LIN {X 0.125,Y -605.700,Z 1096.668,A 0.000,B 0.000,C 90.000,E1 336.230} C_DIS
LIN {X 0.154,Y -607.476,Z 1096.661,A 0.000,B 0.000,C 90.000,E1 334.921} C_DIS
LIN {X -0.038,Y -608.596,Z 1096.655,A 0.000,B 0.000,C 90.000,E1 333.896} C_DIS
LIN {X -0.170,Y -609.283,Z 1096.651,A 0.000,B 0.000,C 90.000,E1 333.127} C_DIS
LIN {X -0.338,Y -609.953,Z 1096.645,A 0.000,B 0.000,C 90.000,E1 332.103} C_DIS
LIN {X -0.253,Y -610.415,Z 1096.638,A 0.000,B 0.000,C 90.000,E1 330.795} C_DIS
LIN {X -0.035,Y -610.410,Z 1096.635,A 0.000,B 0.000,C 90.000,E1 330.255} C_DIS
LIN {X 0.098,Y -609.926,Z 1096.629,A 0.000,B 0.000,C 90.000,E1 329.203} C_DIS
LIN {X 0.317,Y -609.470,Z 1096.626,A 0.000,B 0.000,C 90.000,E1 328.663} C_DIS
LIN {X -0.091,Y -608.172,Z 1096.620,A 0.000,B 0.000,C 90.000,E1 327.661} C_DIS
LIN {X 0.115,Y -607.438,Z 1096.617,A 0.000,B 0.000,C 90.000,E1 327.120} C_DIS
LIN {X 0.003,Y -605.362,Z 1096.612,A 0.000,B 0.000,C 90.000,E1 326.087} C_DIS
LIN {X -0.052,Y -603.766,Z 1096.607,A 0.000,B 0.000,C 90.000,E1 325.308} C_DIS
LIN {X -0.119,Y -602.105,Z 1096.603,A 0.000,B 0.000,C 90.000,E1 324.529} C_DIS
LIN {X 0.286,Y -600.441,Z 1096.599,A 0.000,B 0.000,C 90.000,E1 323.703} C_DIS
LIN {X 0.181,Y -598.723,Z 1096.594,A 0.000,B 0.000,C 90.000,E1 322.924} C_DIS
LIN {X 0.050,Y -595.950,Z 1096.587,A 0.000,B 0.000,C 90.000,E1 321.618} C_DIS
LIN {X 0.006,Y -592.496,Z 1096.578,A 0.000,B 0.000,C 90.000,E1 320.033} C_DIS
LIN {X 0.147,Y -589.672,Z 1096.571,A 0.000,B 0.000,C 90.000,E1 318.690} C_DIS
LIN {X -0.213,Y -586.399,Z 1096.563,A 0.000,B 0.000,C 90.000,E1 317.391} C_DIS
LIN {X -0.034,Y -585.691,Z 1096.562,A 0.000,B 0.000,C 90.000,E1 317.106} C_DIS
LIN {X 0.326,Y -581.328,Z 1096.554,A 0.000,B 0.000,C 90.000,E1 315.729} C_DIS
LIN {X -0.064,Y -578.377,Z 1096.550,A 0.000,B 0.000,C 90.000,E1 314.960} C_DIS
LIN {X -0.234,Y -573.232,Z 1096.542,A 0.000,B 0.000,C 90.000,E1 313.623} C_DIS
LIN {X -0.007,Y -571.099,Z 1096.539,A 0.000,B 0.000,C 90.000,E1 313.056} C_DIS
LIN {X -0.067,Y -567.497,Z 1096.535,A 0.000,B 0.000,C 90.000,E1 312.243} C_DIS
LIN {X -0.132,Y -565.501,Z 1096.532,A 0.000,B 0.000,C 90.000,E1 311.838} C_DIS
LIN {X -0.012,Y -560.708,Z 1096.527,A 0.000,B 0.000,C 90.000,E1 310.862} C_DIS
LIN {X 0.047,Y -555.020,Z 1096.522,A 0.000,B 0.000,C 90.000,E1 309.886} C_DIS
LIN {X 0.086,Y -547.318,Z 1096.515,A 0.000,B 0.000,C 90.000,E1 308.624} C_DIS
LIN {X -0.169,Y -543.344,Z 1096.510,A 0.000,B 0.000,C 90.000,E1 307.810} C_DIS
LIN {X -0.135,Y -542.146,Z 1096.508,A 0.000,B 0.000,C 90.000,E1 307.523} C_DIS
LIN {X -0.102,Y -541.125,Z 1096.507,A 0.000,B 0.000,C 90.000,E1 307.237} C_DIS
LIN {X -0.051,Y -539.374,Z 1096.504,A 0.000,B 0.000,C 90.000,E1 306.664} C_DIS
LIN {X 0.016,Y -537.266,Z 1096.497,A 0.000,B 0.000,C 90.000,E1 305.518} C_DIS
LIN {X 0.039,Y -536.125,Z 1096.493,A 0.000,B 0.000,C 90.000,E1 304.659} C_DIS
LIN {X -0.261,Y -535.957,Z 1096.491,A 0.000,B 0.000,C 90.000,E1 304.405} C_DIS
LIN {X -0.259,Y -535.959,Z 1096.490,A 0.000,B 0.000,C 90.000,E1 304.119} C_DIS
LIN {X 0.039,Y -535.534,Z 1096.487,A 0.000,B 0.000,C 90.000,E1 303.658} C_DIS
LIN {X -0.108,Y -535.459,Z 1096.485,A 0.000,B 0.000,C 90.000,E1 303.245} C_DIS
LIN {X -0.110,Y -535.295,Z 1096.483,A 0.000,B 0.000,C 90.000,E1 302.959} C_DIS
LIN {X -0.116,Y -536.108,Z 1096.469,A 0.000,B 0.000,C 90.000,E1 300.384} C_DIS
LIN {X -0.230,Y -536.522,Z 1096.464,A 0.000,B 0.000,C 90.000,E1 299.539} C_DIS
LIN {X -0.160,Y -537.186,Z 1096.456,A 0.000,B 0.000,C 90.000,E1 298.103} C_DIS
LIN {X 0.124,Y -538.077,Z 1096.447,A 0.000,B 0.000,C 90.000,E1 296.360} C_DIS
LIN {X 0.240,Y -538.580,Z 1096.440,A 0.000,B 0.000,C 90.000,E1 295.207} C_DIS
LIN {X -0.139,Y -539.069,Z 1096.432,A 0.000,B 0.000,C 90.000,E1 293.823} C_DIS
LIN {X -0.271,Y -539.603,Z 1096.421,A 0.000,B 0.000,C 90.000,E1 291.844} C_DIS
LIN {X 0.165,Y -539.876,Z 1096.413,A 0.000,B 0.000,C 90.000,E1 290.375} C_DIS
LIN {X 0.093,Y -539.826,Z 1096.405,A 0.000,B 0.000,C 90.000,E1 288.960} C_DIS
LIN {X 0.125,Y -539.660,Z 1096.399,A 0.000,B 0.000,C 90.000,E1 287.819} C_DIS
LIN {X 0.217,Y -539.404,Z 1096.391,A 0.000,B 0.000,C 90.000,E1 286.386} C_DIS
LIN {X 0.242,Y -539.005,Z 1096.385,A 0.000,B 0.000,C 90.000,E1 285.245} C_DIS
LIN {X 0.242,Y -538.306,Z 1096.375,A 0.000,B 0.000,C 90.000,E1 283.536} C_DIS
LIN {X 0.289,Y -537.333,Z 1096.364,A 0.000,B 0.000,C 90.000,E1 281.535} C_DIS
LIN {X -0.026,Y -536.578,Z 1096.356,A 0.000,B 0.000,C 90.000,E1 280.141} C_DIS
LIN {X 0.240,Y -535.773,Z 1096.347,A 0.000,B 0.000,C 90.000,E1 278.398} C_DIS
LIN {X -0.081,Y -534.772,Z 1096.336,A 0.000,B 0.000,C 90.000,E1 276.429} C_DIS
LIN {X -0.007,Y -533.950,Z 1096.326,A 0.000,B 0.000,C 90.000,E1 274.702} C_DIS
LIN {X -0.005,Y -532.988,Z 1096.315,A 0.000,B 0.000,C 90.000,E1 272.694} C_DIS
LIN {X -0.047,Y -532.085,Z 1096.304,A 0.000,B 0.000,C 90.000,E1 270.688} C_DIS
LIN {X -0.095,Y -531.338,Z 1096.296,A 0.000,B 0.000,C 90.000,E1 269.255} C_DIS
LIN {X -0.133,Y -530.711,Z 1096.289,A 0.000,B 0.000,C 90.000,E1 268.108} C_DIS
LIN {X -0.211,Y -529.719,Z 1096.280,A 0.000,B 0.000,C 90.000,E1 266.388} C_DIS
LIN {X -0.259,Y -528.821,Z 1096.272,A 0.000,B 0.000,C 90.000,E1 264.951} C_DIS
LIN {X 0.195,Y -527.706,Z 1096.264,A 0.000,B 0.000,C 90.000,E1 263.457} C_DIS
LIN {X 0.185,Y -526.825,Z 1096.259,A 0.000,B 0.000,C 90.000,E1 262.591} C_DIS
LIN {X 0.203,Y -525.334,Z 1096.251,A 0.000,B 0.000,C 90.000,E1 261.141} C_DIS
LIN {X 0.243,Y -522.672,Z 1096.236,A 0.000,B 0.000,C 90.000,E1 258.522} C_DIS
LIN {X -0.108,Y -520.672,Z 1096.225,A 0.000,B 0.000,C 90.000,E1 256.520} C_DIS
LIN {X 0.000,Y -519.032,Z 1096.215,A 0.000,B 0.000,C 90.000,E1 254.755} C_DIS
LIN {X -0.159,Y -517.157,Z 1096.206,A 0.000,B 0.000,C 90.000,E1 253.015} C_DIS
LIN {X 0.135,Y -515.263,Z 1096.196,A 0.000,B 0.000,C 90.000,E1 251.221} C_DIS
LIN {X -0.019,Y -513.929,Z 1096.189,A 0.000,B 0.000,C 90.000,E1 250.061} C_DIS
LIN {X 0.048,Y -511.930,Z 1096.179,A 0.000,B 0.000,C 90.000,E1 248.284} C_DIS
LIN {X 0.149,Y -510.140,Z 1096.171,A 0.000,B 0.000,C 90.000,E1 246.794} C_DIS
LIN {X -0.256,Y -507.963,Z 1096.163,A 0.000,B 0.000,C 90.000,E1 245.357} C_DIS
LIN {X -0.120,Y -506.096,Z 1096.156,A 0.000,B 0.000,C 90.000,E1 244.152} C_DIS
LIN {X 0.216,Y -502.642,Z 1096.145,A 0.000,B 0.000,C 90.000,E1 242.025} C_DIS
LIN {X 0.106,Y -500.130,Z 1096.136,A 0.000,B 0.000,C 90.000,E1 240.539} C_DIS
LIN {X -0.242,Y -497.536,Z 1096.128,A 0.000,B 0.000,C 90.000,E1 239.076} C_DIS
LIN {X 0.045,Y -494.892,Z 1096.120,A 0.000,B 0.000,C 90.000,E1 237.533} C_DIS
LIN {X -0.020,Y -491.540,Z 1096.110,A 0.000,B 0.000,C 90.000,E1 235.722} C_DIS
LIN {X 0.168,Y -489.258,Z 1096.103,A 0.000,B 0.000,C 90.000,E1 234.482} C_DIS
LIN {X -0.127,Y -485.664,Z 1096.093,A 0.000,B 0.000,C 90.000,E1 232.683} C_DIS
LIN {X 0.039,Y -483.837,Z 1096.088,A 0.000,B 0.000,C 90.000,E1 231.743} C_DIS
LIN {X 0.179,Y -481.933,Z 1096.082,A 0.000,B 0.000,C 90.000,E1 230.803} C_DIS
LIN {X 0.040,Y -479.438,Z 1096.076,A 0.000,B 0.000,C 90.000,E1 229.585} C_DIS
LIN {X 0.227,Y -475.046,Z 1096.063,A 0.000,B 0.000,C 90.000,E1 227.391} C_DIS
LIN {X -0.082,Y -471.036,Z 1096.051,A 0.000,B 0.000,C 90.000,E1 225.243} C_DIS
LIN {X 0.096,Y -467.602,Z 1096.041,A 0.000,B 0.000,C 90.000,E1 223.338} C_DIS
LIN {X -0.123,Y -464.031,Z 1096.030,A 0.000,B 0.000,C 90.000,E1 221.472} C_DIS
LIN {X -0.082,Y -460.558,Z 1096.020,A 0.000,B 0.000,C 90.000,E1 219.564} C_DIS
LIN {X 0.175,Y -458.294,Z 1096.013,A 0.000,B 0.000,C 90.000,E1 218.257} C_DIS
LIN {X -0.142,Y -454.982,Z 1096.002,A 0.000,B 0.000,C 90.000,E1 216.377} C_DIS
LIN {X 0.108,Y -452.342,Z 1095.993,A 0.000,B 0.000,C 90.000,E1 214.739} C_DIS
LIN {X -0.047,Y -448.715,Z 1095.981,A 0.000,B 0.000,C 90.000,E1 212.498} C_DIS
LIN {X 0.087,Y -444.980,Z 1095.968,A 0.000,B 0.000,C 90.000,E1 210.207} C_DIS
LIN {X 0.267,Y -441.653,Z 1095.955,A 0.000,B 0.000,C 90.000,E1 207.897} C_DIS
LIN {X -0.128,Y -436.875,Z 1095.933,A 0.000,B 0.000,C 90.000,E1 204.003} C_DIS
LIN {X 0.009,Y -435.691,Z 1095.924,A 0.000,B 0.000,C 90.000,E1 202.333} C_DIS
LIN {X -0.094,Y -435.524,Z 1095.919,A 0.000,B 0.000,C 90.000,E1 201.354} C_DIS
LIN {X -0.043,Y -435.962,Z 1095.913,A 0.000,B 0.000,C 90.000,E1 200.355} C_DIS
LIN {X 0.025,Y -436.716,Z 1095.909,A 0.000,B 0.000,C 90.000,E1 199.685} C_DIS
LIN {X -0.046,Y -437.803,Z 1095.906,A 0.000,B 0.000,C 90.000,E1 199.033} C_DIS
LIN {X -0.128,Y -440.135,Z 1095.900,A 0.000,B 0.000,C 90.000,E1 198.055} C_DIS
LIN {X 0.099,Y -443.167,Z 1095.895,A 0.000,B 0.000,C 90.000,E1 197.040} C_DIS
LIN {X -0.038,Y -449.357,Z 1095.886,A 0.000,B 0.000,C 90.000,E1 195.426} C_DIS
LIN {X -0.132,Y -461.079,Z 1095.870,A 0.000,B 0.000,C 90.000,E1 192.703} C_DIS
LIN {X 0.033,Y -472.095,Z 1095.857,A 0.000,B 0.000,C 90.000,E1 190.310} C_DIS
LIN {X -0.084,Y -481.287,Z 1095.847,A 0.000,B 0.000,C 90.000,E1 188.454} C_DIS
LIN {X -0.082,Y -487.906,Z 1095.839,A 0.000,B 0.000,C 90.000,E1 187.068} C_DIS
LIN {X 0.199,Y -495.152,Z 1095.831,A 0.000,B 0.000,C 90.000,E1 185.511} C_DIS
LIN {X -0.011,Y -503.609,Z 1095.821,A 0.000,B 0.000,C 90.000,E1 183.726} C_DIS
LIN {X -0.100,Y -512.003,Z 1095.811,A 0.000,B 0.000,C 90.000,E1 181.949} C_DIS
LIN {X -0.003,Y -520.418,Z 1095.801,A 0.000,B 0.000,C 90.000,E1 180.172} C_DIS
LIN {X 0.022,Y -528.111,Z 1095.792,A 0.000,B 0.000,C 90.000,E1 178.568} C_DIS
LIN {X 0.214,Y -535.794,Z 1095.783,A 0.000,B 0.000,C 90.000,E1 176.963} C_DIS
LIN {X 0.116,Y -544.679,Z 1095.773,A 0.000,B 0.000,C 90.000,E1 175.122} C_DIS
LIN {X -0.004,Y -549.406,Z 1095.768,A 0.000,B 0.000,C 90.000,E1 174.147} C_DIS
LIN {X 0.153,Y -556.789,Z 1095.759,A 0.000,B 0.000,C 90.000,E1 172.591} C_DIS
LIN {X 0.220,Y -563.411,Z 1095.751,A 0.000,B 0.000,C 90.000,E1 171.197} C_DIS
LIN {X -0.146,Y -569.896,Z 1095.744,A 0.000,B 0.000,C 90.000,E1 169.859} C_DIS
LIN {X 0.189,Y -574.291,Z 1095.738,A 0.000,B 0.000,C 90.000,E1 168.870} C_DIS
LIN {X 0.010,Y -578.579,Z 1095.733,A 0.000,B 0.000,C 90.000,E1 167.937} C_DIS
LIN {X -0.232,Y -583.276,Z 1095.727,A 0.000,B 0.000,C 90.000,E1 166.881} C_DIS
LIN {X 0.292,Y -587.790,Z 1095.721,A 0.000,B 0.000,C 90.000,E1 165.755} C_DIS
LIN {X -0.093,Y -591.088,Z 1095.717,A 0.000,B 0.000,C 90.000,E1 164.991} C_DIS
LIN {X -0.026,Y -595.223,Z 1095.711,A 0.000,B 0.000,C 90.000,E1 163.921} C_DIS
LIN {X 0.094,Y -599.082,Z 1095.705,A 0.000,B 0.000,C 90.000,E1 162.851} C_DIS
LIN {X -0.126,Y -602.719,Z 1095.699,A 0.000,B 0.000,C 90.000,E1 161.819} C_DIS
LIN {X 0.281,Y -606.082,Z 1095.693,A 0.000,B 0.000,C 90.000,E1 160.732} C_DIS
LIN {X 0.161,Y -609.317,Z 1095.687,A 0.000,B 0.000,C 90.000,E1 159.699} C_DIS
LIN {X 0.034,Y -613.187,Z 1095.680,A 0.000,B 0.000,C 90.000,E1 158.411} C_DIS
LIN {X -0.065,Y -617.486,Z 1095.672,A 0.000,B 0.000,C 90.000,E1 156.869} C_DIS
LIN {X -0.133,Y -620.262,Z 1095.666,A 0.000,B 0.000,C 90.000,E1 155.845} C_DIS
LIN {X 0.158,Y -624.222,Z 1095.657,A 0.000,B 0.000,C 90.000,E1 154.280} C_DIS
LIN {X 0.196,Y -626.788,Z 1095.652,A 0.000,B 0.000,C 90.000,E1 153.256} C_DIS
LIN {X 0.268,Y -629.156,Z 1095.646,A 0.000,B 0.000,C 90.000,E1 152.231} C_DIS
LIN {X 0.176,Y -632.603,Z 1095.637,A 0.000,B 0.000,C 90.000,E1 150.717} C_DIS
LIN {X 0.117,Y -635.310,Z 1095.630,A 0.000,B 0.000,C 90.000,E1 149.459} C_DIS
LIN {X 0.058,Y -637.475,Z 1095.625,A 0.000,B 0.000,C 90.000,E1 148.456} C_DIS
LIN {X -0.083,Y -640.511,Z 1095.616,A 0.000,B 0.000,C 90.000,E1 146.962} C_DIS
LIN {X -0.174,Y -643.370,Z 1095.608,A 0.000,B 0.000,C 90.000,E1 145.468} C_DIS
LIN {X -0.383,Y -646.173,Z 1095.600,A 0.000,B 0.000,C 90.000,E1 143.989} C_DIS
LIN {X 0.283,Y -649.386,Z 1095.590,A 0.000,B 0.000,C 90.000,E1 142.190} C_DIS
LIN {X 0.040,Y -653.082,Z 1095.579,A 0.000,B 0.000,C 90.000,E1 140.231} C_DIS
LIN {X 0.266,Y -656.480,Z 1095.570,A 0.000,B 0.000,C 90.000,E1 138.485} C_DIS
LIN {X 0.082,Y -659.965,Z 1095.560,A 0.000,B 0.000,C 90.000,E1 136.782} C_DIS
LIN {X -0.069,Y -665.359,Z 1095.546,A 0.000,B 0.000,C 90.000,E1 134.352} C_DIS
LIN {X 0.415,Y -669.544,Z 1095.537,A 0.000,B 0.000,C 90.000,E1 132.609} C_DIS
LIN {X 0.112,Y -674.420,Z 1095.526,A 0.000,B 0.000,C 90.000,E1 130.701} C_DIS
LIN {X 0.042,Y -679.818,Z 1095.514,A 0.000,B 0.000,C 90.000,E1 128.543} C_DIS
LIN {X 0.019,Y -683.572,Z 1095.506,A 0.000,B 0.000,C 90.000,E1 127.111} C_DIS
LIN {X -0.111,Y -686.585,Z 1095.500,A 0.000,B 0.000,C 90.000,E1 125.931} C_DIS
LIN {X -0.079,Y -688.892,Z 1095.494,A 0.000,B 0.000,C 90.000,E1 124.978} C_DIS
LIN {X -0.336,Y -692.370,Z 1095.486,A 0.000,B 0.000,C 90.000,E1 123.579} C_DIS
LIN {X 0.393,Y -695.241,Z 1095.480,A 0.000,B 0.000,C 90.000,E1 122.339} C_DIS
LIN {X -0.163,Y -697.974,Z 1095.473,A 0.000,B 0.000,C 90.000,E1 121.209} C_DIS
LIN {X 0.021,Y -699.867,Z 1095.468,A 0.000,B 0.000,C 90.000,E1 120.256} C_DIS
LIN {X -0.130,Y -701.496,Z 1095.463,A 0.000,B 0.000,C 90.000,E1 119.333} C_DIS
LIN {X 0.354,Y -702.764,Z 1095.458,A 0.000,B 0.000,C 90.000,E1 118.359} C_DIS
LIN {X -0.377,Y -703.513,Z 1095.454,A 0.000,B 0.000,C 90.000,E1 117.719} C_DIS
LIN {X -0.209,Y -704.427,Z 1095.447,A 0.000,B 0.000,C 90.000,E1 116.539} C_DIS
LIN {X -0.004,Y -705.215,Z 1095.442,A 0.000,B 0.000,C 90.000,E1 115.591} C_DIS
LIN {X -0.366,Y -705.443,Z 1095.440,A 0.000,B 0.000,C 90.000,E1 115.155} C_DIS
LIN {X 0.212,Y -705.465,Z 1095.437,A 0.000,B 0.000,C 90.000,E1 114.643} C_DIS
LIN {X -0.144,Y -704.915,Z 1095.434,A 0.000,B 0.000,C 90.000,E1 114.207} C_DIS
LIN {X 0.143,Y -704.559,Z 1095.433,A 0.000,B 0.000,C 90.000,E1 113.951} C_DIS
LIN {X -0.217,Y -702.822,Z 1095.431,A 0.000,B 0.000,C 90.000,E1 113.515} C_DIS
LIN {X 0.062,Y -701.713,Z 1095.429,A 0.000,B 0.000,C 90.000,E1 113.259} C_DIS
LIN {X -0.250,Y -697.898,Z 1095.427,A 0.000,B 0.000,C 90.000,E1 112.823} C_DIS
LIN {X -0.121,Y -696.751,Z 1095.426,A 0.000,B 0.000,C 90.000,E1 112.695} C_DIS
LIN {X -0.259,Y -694.995,Z 1095.425,A 0.000,B 0.000,C 90.000,E1 112.589} C_DIS
LIN {X 0.354,Y -687.350,Z 1095.424,A 0.000,B 0.000,C 90.000,E1 112.206} C_DIS
LIN {X 0.148,Y -685.333,Z 1095.423,A 0.000,B 0.000,C 90.000,E1 112.153} C_DIS
LIN {X -0.094,Y -678.820,Z 1095.423,A 0.000,B 0.000,C 90.000,E1 112.078} C_DIS
LIN {X 0.178,Y -676.366,Z 1095.422,A 0.000,B 0.000,C 90.000,E1 112.025} C_DIS
LIN {X 0.106,Y -604.480,Z 1095.422,A 0.000,B 0.000,C 90.000,E1 112.025} C_DIS
LIN {X -0.075,Y -600.684,Z 1095.421,A 0.000,B 0.000,C 90.000,E1 111.844} C_DIS
LIN {X -0.053,Y -596.181,Z 1095.420,A 0.000,B 0.000,C 90.000,E1 111.535} C_DIS
LIN {X 0.088,Y -587.310,Z 1095.416,A 0.000,B 0.000,C 90.000,E1 110.791} C_DIS
LIN {X -0.171,Y -576.224,Z 1095.410,A 0.000,B 0.000,C 90.000,E1 109.866} C_DIS
LIN {X -0.191,Y -573.211,Z 1095.409,A 0.000,B 0.000,C 90.000,E1 109.631} C_DIS
LIN {X 0.083,Y -568.673,Z 1095.407,A 0.000,B 0.000,C 90.000,E1 109.268} C_DIS
LIN {X -0.149,Y -560.368,Z 1095.404,A 0.000,B 0.000,C 90.000,E1 108.779} C_DIS
LIN {X 0.265,Y -553.965,Z 1095.402,A 0.000,B 0.000,C 90.000,E1 108.362} C_DIS
LIN {X 0.272,Y -549.698,Z 1095.401,A 0.000,B 0.000,C 90.000,E1 108.055} C_DIS
LIN {X 0.131,Y -548.304,Z 1095.399,A 0.000,B 0.000,C 90.000,E1 107.873} C_DIS
LIN {X 0.090,Y -548.287,Z 1095.399,A 0.000,B 0.000,C 90.000,E1 107.873} C_DIS
LIN {X 0.127,Y -547.923,Z 1095.397,A 0.000,B 0.000,C 90.000,E1 107.457} C_DIS
LIN {X 0.056,Y -548.040,Z 1095.394,A 0.000,B 0.000,C 90.000,E1 106.985} C_DIS
LIN {X 0.214,Y -548.793,Z 1095.388,A 0.000,B 0.000,C 90.000,E1 105.843} C_DIS
LIN {X 0.147,Y -550.159,Z 1095.377,A 0.000,B 0.000,C 90.000,E1 103.883} C_DIS
LIN {X 0.094,Y -552.366,Z 1095.363,A 0.000,B 0.000,C 90.000,E1 101.366} C_DIS
LIN {X -0.112,Y -554.617,Z 1095.351,A 0.000,B 0.000,C 90.000,E1 99.151} C_DIS
LIN {X 0.012,Y -556.374,Z 1095.342,A 0.000,B 0.000,C 90.000,E1 97.466} C_DIS
LIN {X 0.024,Y -558.186,Z 1095.332,A 0.000,B 0.000,C 90.000,E1 95.796} C_DIS
LIN {X -0.132,Y -559.241,Z 1095.326,A 0.000,B 0.000,C 90.000,E1 94.702} C_DIS
LIN {X -0.230,Y -560.255,Z 1095.318,A 0.000,B 0.000,C 90.000,E1 93.326} C_DIS
LIN {X -0.189,Y -561.182,Z 1095.309,A 0.000,B 0.000,C 90.000,E1 91.661} C_DIS
LIN {X 0.197,Y -561.767,Z 1095.303,A 0.000,B 0.000,C 90.000,E1 90.516} C_DIS
LIN {X 0.236,Y -562.529,Z 1095.294,A 0.000,B 0.000,C 90.000,E1 88.854} C_DIS
LIN {X 0.199,Y -563.140,Z 1095.286,A 0.000,B 0.000,C 90.000,E1 87.478} C_DIS
LIN {X 0.171,Y -563.693,Z 1095.278,A 0.000,B 0.000,C 90.000,E1 86.102} C_DIS
LIN {X 0.187,Y -564.289,Z 1095.271,A 0.000,B 0.000,C 90.000,E1 84.723} C_DIS
LIN {X -0.040,Y -564.909,Z 1095.260,A 0.000,B 0.000,C 90.000,E1 82.818} C_DIS
LIN {X 0.059,Y -565.402,Z 1095.252,A 0.000,B 0.000,C 90.000,E1 81.432} C_DIS
LIN {X 0.203,Y -566.285,Z 1095.240,A 0.000,B 0.000,C 90.000,E1 79.218} C_DIS
LIN {X 0.192,Y -567.149,Z 1095.230,A 0.000,B 0.000,C 90.000,E1 77.297} C_DIS
LIN {X -0.112,Y -568.186,Z 1095.219,A 0.000,B 0.000,C 90.000,E1 75.408} C_DIS
LIN {X 0.133,Y -569.223,Z 1095.210,A 0.000,B 0.000,C 90.000,E1 73.740} C_DIS
LIN {X 0.198,Y -570.707,Z 1095.199,A 0.000,B 0.000,C 90.000,E1 71.819} C_DIS
LIN {X 0.102,Y -572.578,Z 1095.187,A 0.000,B 0.000,C 90.000,E1 69.645} C_DIS
LIN {X -0.267,Y -573.564,Z 1095.181,A 0.000,B 0.000,C 90.000,E1 68.592} C_DIS
LIN {X 0.119,Y -574.962,Z 1095.172,A 0.000,B 0.000,C 90.000,E1 66.922} C_DIS
LIN {X -0.004,Y -576.261,Z 1095.163,A 0.000,B 0.000,C 90.000,E1 65.305} C_DIS
LIN {X 0.160,Y -577.020,Z 1095.157,A 0.000,B 0.000,C 90.000,E1 64.204} C_DIS
LIN {X -0.056,Y -577.982,Z 1095.149,A 0.000,B 0.000,C 90.000,E1 62.871} C_DIS
LIN {X -0.144,Y -579.004,Z 1095.140,A 0.000,B 0.000,C 90.000,E1 61.257} C_DIS
LIN {X -0.295,Y -579.526,Z 1095.136,A 0.000,B 0.000,C 90.000,E1 60.461} C_DIS
LIN {X 0.073,Y -580.527,Z 1095.125,A 0.000,B 0.000,C 90.000,E1 58.535} C_DIS
LIN {X -0.054,Y -581.273,Z 1095.118,A 0.000,B 0.000,C 90.000,E1 57.199} C_DIS
LIN {X -0.173,Y -582.080,Z 1095.109,A 0.000,B 0.000,C 90.000,E1 55.595} C_DIS
LIN {X -0.269,Y -582.743,Z 1095.100,A 0.000,B 0.000,C 90.000,E1 53.989} C_DIS
LIN {X 0.265,Y -583.037,Z 1095.095,A 0.000,B 0.000,C 90.000,E1 53.130} C_DIS
LIN {X 0.164,Y -583.296,Z 1095.089,A 0.000,B 0.000,C 90.000,E1 52.065} C_DIS
LIN {X 0.244,Y -583.440,Z 1095.085,A 0.000,B 0.000,C 90.000,E1 51.251} C_DIS
LIN {X 0.054,Y -583.375,Z 1095.079,A 0.000,B 0.000,C 90.000,E1 50.194} C_DIS
LIN {X 0.044,Y -583.124,Z 1095.072,A 0.000,B 0.000,C 90.000,E1 48.852} C_DIS
LIN {X -0.024,Y -582.658,Z 1095.064,A 0.000,B 0.000,C 90.000,E1 47.514} C_DIS
LIN {X 0.329,Y -582.067,Z 1095.057,A 0.000,B 0.000,C 90.000,E1 46.134} C_DIS
LIN {X 0.092,Y -581.478,Z 1095.051,A 0.000,B 0.000,C 90.000,E1 45.081} C_DIS
LIN {X -0.154,Y -580.614,Z 1095.045,A 0.000,B 0.000,C 90.000,E1 44.028} C_DIS
LIN {X -0.267,Y -579.161,Z 1095.037,A 0.000,B 0.000,C 90.000,E1 42.690} C_DIS
LIN {X 0.150,Y -578.176,Z 1095.033,A 0.000,B 0.000,C 90.000,E1 41.838} C_DIS
LIN {X -0.111,Y -576.543,Z 1095.027,A 0.000,B 0.000,C 90.000,E1 40.782} C_DIS
LIN {X -0.023,Y -574.782,Z 1095.021,A 0.000,B 0.000,C 90.000,E1 39.688} C_DIS
LIN {X 0.105,Y -572.677,Z 1095.015,A 0.000,B 0.000,C 90.000,E1 38.588} C_DIS
LIN {X 0.032,Y -571.505,Z 1095.011,A 0.000,B 0.000,C 90.000,E1 38.051} C_DIS
LIN {X 0.121,Y -568.854,Z 1095.005,A 0.000,B 0.000,C 90.000,E1 36.950} C_DIS
LIN {X 0.040,Y -566.430,Z 1095.001,A 0.000,B 0.000,C 90.000,E1 36.137} C_DIS
LIN {X 0.057,Y -563.702,Z 1094.996,A 0.000,B 0.000,C 90.000,E1 35.311} C_DIS
LIN {X 0.165,Y -562.776,Z 1094.995,A 0.000,B 0.000,C 90.000,E1 35.025} C_DIS
LIN {X 0.148,Y -559.473,Z 1094.990,A 0.000,B 0.000,C 90.000,E1 34.199} C_DIS
LIN {X 0.098,Y -555.824,Z 1094.985,A 0.000,B 0.000,C 90.000,E1 33.372} C_DIS
LIN {X -0.116,Y -551.249,Z 1094.980,A 0.000,B 0.000,C 90.000,E1 32.418} C_DIS
LIN {X -0.138,Y -547.615,Z 1094.976,A 0.000,B 0.000,C 90.000,E1 31.720} C_DIS
LIN {X 0.006,Y -542.293,Z 1094.971,A 0.000,B 0.000,C 90.000,E1 30.718} C_DIS
LIN {X 0.217,Y -539.034,Z 1094.968,A 0.000,B 0.000,C 90.000,E1 30.129} C_DIS
LIN {X 0.125,Y -533.734,Z 1094.963,A 0.000,B 0.000,C 90.000,E1 29.283} C_DIS
LIN {X -0.189,Y -529.885,Z 1094.960,A 0.000,B 0.000,C 90.000,E1 28.743} C_DIS
LIN {X 0.245,Y -524.730,Z 1094.956,A 0.000,B 0.000,C 90.000,E1 27.975} C_DIS
LIN {X 0.163,Y -519.113,Z 1094.952,A 0.000,B 0.000,C 90.000,E1 27.257} C_DIS
LIN {X -0.033,Y -514.260,Z 1094.948,A 0.000,B 0.000,C 90.000,E1 26.693} C_DIS
LIN {X 0.144,Y -510.354,Z 1094.946,A 0.000,B 0.000,C 90.000,E1 26.232} C_DIS
LIN {X -0.143,Y -501.323,Z 1094.940,A 0.000,B 0.000,C 90.000,E1 25.283} C_DIS
LIN {X 0.202,Y -491.734,Z 1094.935,A 0.000,B 0.000,C 90.000,E1 24.259} C_DIS
LIN {X -0.175,Y -480.169,Z 1094.929,A 0.000,B 0.000,C 90.000,E1 23.206} C_DIS
LIN {X -0.059,Y -471.195,Z 1094.924,A 0.000,B 0.000,C 90.000,E1 22.386} C_DIS
LIN {X 0.121,Y -462.308,Z 1094.920,A 0.000,B 0.000,C 90.000,E1 21.589} C_DIS
LIN {X -0.196,Y -447.285,Z 1094.913,A 0.000,B 0.000,C 90.000,E1 20.301} C_DIS
LIN {X 0.058,Y -432.704,Z 1094.905,A 0.000,B 0.000,C 90.000,E1 18.906} C_DIS
LIN {X 0.131,Y -419.955,Z 1094.898,A 0.000,B 0.000,C 90.000,E1 17.583} C_DIS
LIN {X -0.238,Y -407.659,Z 1094.890,A 0.000,B 0.000,C 90.000,E1 16.205} C_DIS
LIN {X -0.087,Y -400.049,Z 1094.884,A 0.000,B 0.000,C 90.000,E1 15.190} C_DIS
LIN {X -0.031,Y -396.972,Z 1094.882,A 0.000,B 0.000,C 90.000,E1 14.717} C_DIS
LIN {X 0.091,Y -394.672,Z 1094.879,A 0.000,B 0.000,C 90.000,E1 14.245} C_DIS
LIN {X 0.121,Y -393.899,Z 1094.878,A 0.000,B 0.000,C 90.000,E1 14.064} C_DIS
LIN {X -0.118,Y -392.407,Z 1094.875,A 0.000,B 0.000,C 90.000,E1 13.467} C_DIS
LIN {X 0.010,Y -392.071,Z 1094.871,A 0.000,B 0.000,C 90.000,E1 12.827} C_DIS
LIN {X -0.067,Y -392.700,Z 1094.866,A 0.000,B 0.000,C 90.000,E1 11.951} C_DIS
LIN {X -0.076,Y -393.650,Z 1094.862,A 0.000,B 0.000,C 90.000,E1 11.243} C_DIS
LIN {X 0.058,Y -399.036,Z 1094.847,A 0.000,B 0.000,C 90.000,E1 8.398} C_DIS
LIN {X -0.076,Y -403.886,Z 1094.835,A 0.000,B 0.000,C 90.000,E1 6.315} C_DIS
LIN {X -0.144,Y -406.801,Z 1094.828,A 0.000,B 0.000,C 90.000,E1 5.106} C_DIS
LIN {X -0.069,Y -409.121,Z 1094.825,A 0.000,B 0.000,C 90.000,E1 4.473} C_DIS
LIN {X -0.082,Y -409.916,Z 1094.824,A 0.000,B 0.000,C 90.000,E1 4.302} C_DIS
LIN {X 0.116,Y -412.164,Z 1094.822,A 0.000,B 0.000,C 90.000,E1 3.898} C_DIS
LIN {X 0.164,Y -415.347,Z 1094.820,A 0.000,B 0.000,C 90.000,E1 3.555} C_DIS
LIN {X -0.109,Y -416.999,Z 1094.819,A 0.000,B 0.000,C 90.000,E1 3.440} C_DIS
LIN {X 0.097,Y -425.569,Z 1094.816,A 0.000,B 0.000,C 90.000,E1 2.808} C_DIS
LIN {X -0.175,Y -443.340,Z 1094.809,A 0.000,B 0.000,C 90.000,E1 1.661} C_DIS
LIN {X 0.080,Y -466.189,Z 1094.801,A 0.000,B 0.000,C 90.000,E1 0.172} C_DIS
LIN {X -0.037,Y -477.380,Z 1094.797,A 0.000,B 0.000,C 90.000,E1 359.484} C_DIS
LIN {X 0.024,Y -487.011,Z 1094.794,A 0.000,B 0.000,C 90.000,E1 358.854} C_DIS
LIN {X -0.051,Y -496.530,Z 1094.790,A 0.000,B 0.000,C 90.000,E1 358.224} C_DIS
LIN {X 0.147,Y -504.195,Z 1094.787,A 0.000,B 0.000,C 90.000,E1 357.650} C_DIS
LIN {X 0.101,Y -510.302,Z 1094.785,A 0.000,B 0.000,C 90.000,E1 357.192} C_DIS
LIN {X -0.127,Y -517.564,Z 1094.781,A 0.000,B 0.000,C 90.000,E1 356.617} C_DIS
LIN {X 0.114,Y -523.135,Z 1094.778,A 0.000,B 0.000,C 90.000,E1 356.102} C_DIS
LIN {X 0.083,Y -528.569,Z 1094.776,A 0.000,B 0.000,C 90.000,E1 355.584} C_DIS
LIN {X -0.069,Y -534.715,Z 1094.772,A 0.000,B 0.000,C 90.000,E1 354.951} C_DIS
LIN {X -0.215,Y -540.710,Z 1094.768,A 0.000,B 0.000,C 90.000,E1 354.261} C_DIS
LIN {X -0.144,Y -545.153,Z 1094.765,A 0.000,B 0.000,C 90.000,E1 353.685} C_DIS
LIN {X -0.043,Y -549.285,Z 1094.762,A 0.000,B 0.000,C 90.000,E1 353.109} C_DIS
LIN {X -0.095,Y -553.822,Z 1094.758,A 0.000,B 0.000,C 90.000,E1 352.413} C_DIS
LIN {X 0.069,Y -557.160,Z 1094.755,A 0.000,B 0.000,C 90.000,E1 351.837} C_DIS
LIN {X 0.092,Y -560.836,Z 1094.751,A 0.000,B 0.000,C 90.000,E1 351.141} C_DIS
LIN {X 0.149,Y -564.192,Z 1094.747,A 0.000,B 0.000,C 90.000,E1 350.443} C_DIS
LIN {X 0.169,Y -569.015,Z 1094.741,A 0.000,B 0.000,C 90.000,E1 349.342} C_DIS
LIN {X -0.211,Y -573.366,Z 1094.735,A 0.000,B 0.000,C 90.000,E1 348.285} C_DIS
LIN {X 0.035,Y -577.311,Z 1094.729,A 0.000,B 0.000,C 90.000,E1 347.173} C_DIS
LIN {X -0.011,Y -581.876,Z 1094.721,A 0.000,B 0.000,C 90.000,E1 345.825} C_DIS
LIN {X -0.076,Y -585.368,Z 1094.715,A 0.000,B 0.000,C 90.000,E1 344.755} C_DIS
LIN {X 0.319,Y -589.432,Z 1094.708,A 0.000,B 0.000,C 90.000,E1 343.378} C_DIS
LIN {X 0.229,Y -593.386,Z 1094.700,A 0.000,B 0.000,C 90.000,E1 342.054} C_DIS
LIN {X 0.057,Y -595.686,Z 1094.696,A 0.000,B 0.000,C 90.000,E1 341.275} C_DIS
LIN {X -0.101,Y -597.731,Z 1094.692,A 0.000,B 0.000,C 90.000,E1 340.496} C_DIS
LIN {X 0.046,Y -601.413,Z 1094.683,A 0.000,B 0.000,C 90.000,E1 338.901} C_DIS
LIN {X 0.077,Y -603.488,Z 1094.677,A 0.000,B 0.000,C 90.000,E1 337.847} C_DIS
LIN {X 0.138,Y -605.343,Z 1094.671,A 0.000,B 0.000,C 90.000,E1 336.794} C_DIS
LIN {X 0.217,Y -606.869,Z 1094.665,A 0.000,B 0.000,C 90.000,E1 335.741} C_DIS
LIN {X 0.015,Y -608.275,Z 1094.660,A 0.000,B 0.000,C 90.000,E1 334.717} C_DIS
LIN {X 0.344,Y -609.636,Z 1094.652,A 0.000,B 0.000,C 90.000,E1 333.384} C_DIS
LIN {X 0.142,Y -610.579,Z 1094.645,A 0.000,B 0.000,C 90.000,E1 332.103} C_DIS
LIN {X 0.238,Y -611.118,Z 1094.638,A 0.000,B 0.000,C 90.000,E1 330.795} C_DIS
LIN {X -0.109,Y -611.116,Z 1094.634,A 0.000,B 0.000,C 90.000,E1 330.049} C_DIS
LIN {X 0.037,Y -610.619,Z 1094.628,A 0.000,B 0.000,C 90.000,E1 328.997} C_DIS
LIN {X -0.355,Y -609.613,Z 1094.622,A 0.000,B 0.000,C 90.000,E1 327.995} C_DIS
LIN {X 0.135,Y -608.605,Z 1094.618,A 0.000,B 0.000,C 90.000,E1 327.168} C_DIS
LIN {X 0.044,Y -606.732,Z 1094.612,A 0.000,B 0.000,C 90.000,E1 326.135} C_DIS
LIN {X -0.073,Y -604.667,Z 1094.606,A 0.000,B 0.000,C 90.000,E1 325.102} C_DIS
LIN {X 0.102,Y -603.685,Z 1094.603,A 0.000,B 0.000,C 90.000,E1 324.562} C_DIS
LIN {X -0.224,Y -602.611,Z 1094.600,A 0.000,B 0.000,C 90.000,E1 324.069} C_DIS
LIN {X 0.030,Y -602.172,Z 1094.599,A 0.000,B 0.000,C 90.000,E1 323.783} C_DIS
LIN {X 0.052,Y -601.085,Z 1094.596,A 0.000,B 0.000,C 90.000,E1 323.256} C_DIS
LIN {X -0.058,Y -600.623,Z 1094.594,A 0.000,B 0.000,C 90.000,E1 323.004} C_DIS
LIN {X 0.078,Y -597.509,Z 1094.586,A 0.000,B 0.000,C 90.000,E1 321.412} C_DIS
LIN {X 0.046,Y -593.409,Z 1094.574,A 0.000,B 0.000,C 90.000,E1 319.299} C_DIS
LIN {X 0.231,Y -591.841,Z 1094.570,A 0.000,B 0.000,C 90.000,E1 318.485} C_DIS
LIN {X -0.289,Y -589.478,Z 1094.564,A 0.000,B 0.000,C 90.000,E1 317.472} C_DIS
LIN {X 0.241,Y -587.370,Z 1094.559,A 0.000,B 0.000,C 90.000,E1 316.620} C_DIS
LIN {X -0.256,Y -585.863,Z 1094.556,A 0.000,B 0.000,C 90.000,E1 316.134} C_DIS
LIN {X 0.118,Y -581.725,Z 1094.549,A 0.000,B 0.000,C 90.000,E1 314.757} C_DIS
LIN {X -0.005,Y -579.818,Z 1094.546,A 0.000,B 0.000,C 90.000,E1 314.231} C_DIS
LIN {X 0.014,Y -577.222,Z 1094.541,A 0.000,B 0.000,C 90.000,E1 313.419} C_DIS
LIN {X 0.132,Y -576.196,Z 1094.540,A 0.000,B 0.000,C 90.000,E1 313.137} C_DIS
LIN {X 0.125,Y -573.480,Z 1094.535,A 0.000,B 0.000,C 90.000,E1 312.324} C_DIS
LIN {X 0.350,Y -571.342,Z 1094.532,A 0.000,B 0.000,C 90.000,E1 311.757} C_DIS
LIN {X 0.116,Y -567.147,Z 1094.527,A 0.000,B 0.000,C 90.000,E1 310.825} C_DIS
LIN {X -0.215,Y -563.829,Z 1094.523,A 0.000,B 0.000,C 90.000,E1 310.172} C_DIS
LIN {X 0.014,Y -559.175,Z 1094.519,A 0.000,B 0.000,C 90.000,E1 309.322} C_DIS
LIN {X -0.109,Y -548.365,Z 1094.508,A 0.000,B 0.000,C 90.000,E1 307.523} C_DIS
LIN {X -0.008,Y -545.425,Z 1094.505,A 0.000,B 0.000,C 90.000,E1 306.950} C_DIS
LIN {X 0.216,Y -543.674,Z 1094.503,A 0.000,B 0.000,C 90.000,E1 306.503} C_DIS
LIN {X 0.252,Y -542.415,Z 1094.501,A 0.000,B 0.000,C 90.000,E1 306.217} C_DIS
LIN {X -0.070,Y -541.014,Z 1094.499,A 0.000,B 0.000,C 90.000,E1 305.724} C_DIS
LIN {X -0.046,Y -540.037,Z 1094.497,A 0.000,B 0.000,C 90.000,E1 305.438} C_DIS
LIN {X -0.008,Y -538.526,Z 1094.494,A 0.000,B 0.000,C 90.000,E1 304.865} C_DIS
LIN {X -0.167,Y -537.743,Z 1094.491,A 0.000,B 0.000,C 90.000,E1 304.405} C_DIS
LIN {X -0.157,Y -537.629,Z 1094.490,A 0.000,B 0.000,C 90.000,E1 304.119} C_DIS
LIN {X 0.152,Y -536.931,Z 1094.487,A 0.000,B 0.000,C 90.000,E1 303.658} C_DIS
LIN {X -0.370,Y -536.760,Z 1094.485,A 0.000,B 0.000,C 90.000,E1 303.372} C_DIS
LIN {X 0.229,Y -536.334,Z 1094.483,A 0.000,B 0.000,C 90.000,E1 302.880} C_DIS
LIN {X 0.083,Y -536.359,Z 1094.480,A 0.000,B 0.000,C 90.000,E1 302.467} C_DIS
LIN {X -0.207,Y -536.161,Z 1094.479,A 0.000,B 0.000,C 90.000,E1 302.212} C_DIS
LIN {X 0.121,Y -536.268,Z 1094.471,A 0.000,B 0.000,C 90.000,E1 300.747} C_DIS
LIN {X -0.170,Y -536.584,Z 1094.468,A 0.000,B 0.000,C 90.000,E1 300.207} C_DIS
LIN {X 0.082,Y -537.323,Z 1094.457,A 0.000,B 0.000,C 90.000,E1 298.180} C_DIS
LIN {X 0.106,Y -538.360,Z 1094.446,A 0.000,B 0.000,C 90.000,E1 296.181} C_DIS
LIN {X -0.040,Y -538.952,Z 1094.438,A 0.000,B 0.000,C 90.000,E1 294.771} C_DIS
LIN {X 0.084,Y -539.387,Z 1094.430,A 0.000,B 0.000,C 90.000,E1 293.334} C_DIS
LIN {X -0.061,Y -539.858,Z 1094.420,A 0.000,B 0.000,C 90.000,E1 291.642} C_DIS
LIN {X 0.144,Y -540.136,Z 1094.414,A 0.000,B 0.000,C 90.000,E1 290.482} C_DIS
LIN {X -0.109,Y -540.115,Z 1094.406,A 0.000,B 0.000,C 90.000,E1 289.087} C_DIS
LIN {X -0.068,Y -539.983,Z 1094.400,A 0.000,B 0.000,C 90.000,E1 287.946} C_DIS
LIN {X 0.188,Y -539.736,Z 1094.392,A 0.000,B 0.000,C 90.000,E1 286.496} C_DIS
LIN {X 0.068,Y -539.366,Z 1094.385,A 0.000,B 0.000,C 90.000,E1 285.371} C_DIS
LIN {X 0.211,Y -538.697,Z 1094.376,A 0.000,B 0.000,C 90.000,E1 283.647} C_DIS
LIN {X 0.151,Y -537.736,Z 1094.365,A 0.000,B 0.000,C 90.000,E1 281.658} C_DIS
LIN {X 0.069,Y -536.717,Z 1094.354,A 0.000,B 0.000,C 90.000,E1 279.670} C_DIS
LIN {X 0.271,Y -536.000,Z 1094.346,A 0.000,B 0.000,C 90.000,E1 278.219} C_DIS
LIN {X -0.099,Y -535.145,Z 1094.336,A 0.000,B 0.000,C 90.000,E1 276.543} C_DIS
LIN {X -0.065,Y -534.319,Z 1094.327,A 0.000,B 0.000,C 90.000,E1 274.821} C_DIS
LIN {X -0.012,Y -533.345,Z 1094.316,A 0.000,B 0.000,C 90.000,E1 272.808} C_DIS
LIN {X -0.053,Y -532.330,Z 1094.303,A 0.000,B 0.000,C 90.000,E1 270.516} C_DIS
LIN {X -0.122,Y -531.281,Z 1094.292,A 0.000,B 0.000,C 90.000,E1 268.511} C_DIS
LIN {X -0.188,Y -530.108,Z 1094.281,A 0.000,B 0.000,C 90.000,E1 266.502} C_DIS
LIN {X -0.229,Y -529.207,Z 1094.272,A 0.000,B 0.000,C 90.000,E1 265.065} C_DIS
LIN {X 0.236,Y -528.103,Z 1094.265,A 0.000,B 0.000,C 90.000,E1 263.571} C_DIS
LIN {X 0.233,Y -527.250,Z 1094.260,A 0.000,B 0.000,C 90.000,E1 262.704} C_DIS
LIN {X 0.198,Y -525.447,Z 1094.250,A 0.000,B 0.000,C 90.000,E1 260.971} C_DIS
LIN {X -0.178,Y -522.771,Z 1094.235,A 0.000,B 0.000,C 90.000,E1 258.398} C_DIS
LIN {X -0.132,Y -521.060,Z 1094.226,A 0.000,B 0.000,C 90.000,E1 256.645} C_DIS
LIN {X 0.113,Y -519.397,Z 1094.216,A 0.000,B 0.000,C 90.000,E1 254.866} C_DIS
LIN {X -0.050,Y -517.208,Z 1094.205,A 0.000,B 0.000,C 90.000,E1 252.834} C_DIS
LIN {X -0.244,Y -515.325,Z 1094.195,A 0.000,B 0.000,C 90.000,E1 251.094} C_DIS
LIN {X -0.142,Y -513.335,Z 1094.185,A 0.000,B 0.000,C 90.000,E1 249.316} C_DIS
LIN {X -0.201,Y -511.616,Z 1094.177,A 0.000,B 0.000,C 90.000,E1 247.847} C_DIS
LIN {X -0.215,Y -510.155,Z 1094.170,A 0.000,B 0.000,C 90.000,E1 246.666} C_DIS
LIN {X 0.058,Y -507.948,Z 1094.162,A 0.000,B 0.000,C 90.000,E1 245.153} C_DIS
LIN {X -0.024,Y -506.049,Z 1094.155,A 0.000,B 0.000,C 90.000,E1 243.973} C_DIS
LIN {X -0.143,Y -502.602,Z 1094.144,A 0.000,B 0.000,C 90.000,E1 241.897} C_DIS
LIN {X 0.040,Y -499.537,Z 1094.134,A 0.000,B 0.000,C 90.000,E1 240.078} C_DIS
LIN {X -0.061,Y -496.971,Z 1094.125,A 0.000,B 0.000,C 90.000,E1 238.584} C_DIS
LIN {X -0.052,Y -494.771,Z 1094.119,A 0.000,B 0.000,C 90.000,E1 237.375} C_DIS
LIN {X 0.019,Y -491.362,Z 1094.109,A 0.000,B 0.000,C 90.000,E1 235.548} C_DIS
LIN {X 0.081,Y -489.063,Z 1094.102,A 0.000,B 0.000,C 90.000,E1 234.322} C_DIS
LIN {X 0.175,Y -485.462,Z 1094.092,A 0.000,B 0.000,C 90.000,E1 232.477} C_DIS
LIN {X -0.043,Y -483.593,Z 1094.087,A 0.000,B 0.000,C 90.000,E1 231.582} C_DIS
LIN {X 0.029,Y -480.473,Z 1094.078,A 0.000,B 0.000,C 90.000,E1 230.033} C_DIS
LIN {X 0.141,Y -476.640,Z 1094.068,A 0.000,B 0.000,C 90.000,E1 228.162} C_DIS
LIN {X -0.266,Y -471.339,Z 1094.052,A 0.000,B 0.000,C 90.000,E1 225.405} C_DIS
LIN {X 0.165,Y -468.492,Z 1094.043,A 0.000,B 0.000,C 90.000,E1 223.785} C_DIS
LIN {X -0.039,Y -464.934,Z 1094.033,A 0.000,B 0.000,C 90.000,E1 221.919} C_DIS
LIN {X -0.234,Y -460.835,Z 1094.021,A 0.000,B 0.000,C 90.000,E1 219.725} C_DIS
LIN {X 0.031,Y -458.529,Z 1094.014,A 0.000,B 0.000,C 90.000,E1 218.418} C_DIS
LIN {X -0.004,Y -455.185,Z 1094.003,A 0.000,B 0.000,C 90.000,E1 216.503} C_DIS
LIN {X 0.075,Y -451.910,Z 1093.992,A 0.000,B 0.000,C 90.000,E1 214.565} C_DIS
LIN {X 0.085,Y -448.743,Z 1093.981,A 0.000,B 0.000,C 90.000,E1 212.625} C_DIS
LIN {X 0.214,Y -444.927,Z 1093.969,A 0.000,B 0.000,C 90.000,E1 210.335} C_DIS
LIN {X -0.209,Y -441.492,Z 1093.956,A 0.000,B 0.000,C 90.000,E1 208.103} C_DIS
LIN {X -0.032,Y -436.717,Z 1093.936,A 0.000,B 0.000,C 90.000,E1 204.463} C_DIS
LIN {X 0.108,Y -434.914,Z 1093.925,A 0.000,B 0.000,C 90.000,E1 202.461} C_DIS
LIN {X -0.017,Y -434.558,Z 1093.918,A 0.000,B 0.000,C 90.000,E1 201.153} C_DIS
LIN {X -0.135,Y -434.902,Z 1093.912,A 0.000,B 0.000,C 90.000,E1 200.174} C_DIS
LIN {X -0.076,Y -435.642,Z 1093.908,A 0.000,B 0.000,C 90.000,E1 199.504} C_DIS
LIN {X -0.155,Y -436.730,Z 1093.905,A 0.000,B 0.000,C 90.000,E1 198.852} C_DIS
LIN {X 0.167,Y -439.025,Z 1093.899,A 0.000,B 0.000,C 90.000,E1 197.819} C_DIS
LIN {X -0.039,Y -442.124,Z 1093.894,A 0.000,B 0.000,C 90.000,E1 196.858} C_DIS
LIN {X -0.196,Y -448.430,Z 1093.885,A 0.000,B 0.000,C 90.000,E1 195.245} C_DIS
LIN {X 0.187,Y -461.114,Z 1093.869,A 0.000,B 0.000,C 90.000,E1 192.299} C_DIS
LIN {X 0.012,Y -473.171,Z 1093.854,A 0.000,B 0.000,C 90.000,E1 189.792} C_DIS
LIN {X 0.144,Y -480.972,Z 1093.846,A 0.000,B 0.000,C 90.000,E1 188.219} C_DIS
LIN {X 0.139,Y -487.642,Z 1093.838,A 0.000,B 0.000,C 90.000,E1 186.834} C_DIS
LIN {X 0.196,Y -494.224,Z 1093.830,A 0.000,B 0.000,C 90.000,E1 185.454} C_DIS
LIN {X -0.166,Y -498.489,Z 1093.825,A 0.000,B 0.000,C 90.000,E1 184.588} C_DIS
LIN {X -0.153,Y -504.197,Z 1093.819,A 0.000,B 0.000,C 90.000,E1 183.383} C_DIS
LIN {X -0.211,Y -512.704,Z 1093.809,A 0.000,B 0.000,C 90.000,E1 181.604} C_DIS
LIN {X 0.174,Y -520.461,Z 1093.800,A 0.000,B 0.000,C 90.000,E1 179.943} C_DIS
LIN {X 0.203,Y -528.245,Z 1093.791,A 0.000,B 0.000,C 90.000,E1 178.339} C_DIS
LIN {X -0.108,Y -535.965,Z 1093.782,A 0.000,B 0.000,C 90.000,E1 176.788} C_DIS
LIN {X -0.240,Y -544.904,Z 1093.772,A 0.000,B 0.000,C 90.000,E1 174.951} C_DIS
LIN {X 0.242,Y -549.666,Z 1093.766,A 0.000,B 0.000,C 90.000,E1 173.913} C_DIS
LIN {X -0.260,Y -555.760,Z 1093.759,A 0.000,B 0.000,C 90.000,E1 172.704} C_DIS
LIN {X -0.214,Y -562.455,Z 1093.752,A 0.000,B 0.000,C 90.000,E1 171.310} C_DIS
LIN {X 0.105,Y -568.336,Z 1093.745,A 0.000,B 0.000,C 90.000,E1 170.038} C_DIS
LIN {X 0.051,Y -574.035,Z 1093.738,A 0.000,B 0.000,C 90.000,E1 168.814} C_DIS
LIN {X -0.247,Y -578.900,Z 1093.732,A 0.000,B 0.000,C 90.000,E1 167.757} C_DIS
LIN {X 0.083,Y -583.624,Z 1093.726,A 0.000,B 0.000,C 90.000,E1 166.645} C_DIS
LIN {X 0.297,Y -589.282,Z 1093.719,A 0.000,B 0.000,C 90.000,E1 165.283} C_DIS
LIN {X 0.040,Y -594.552,Z 1093.711,A 0.000,B 0.000,C 90.000,E1 163.976} C_DIS
LIN {X 0.155,Y -598.457,Z 1093.705,A 0.000,B 0.000,C 90.000,E1 162.906} C_DIS
LIN {X -0.071,Y -602.117,Z 1093.699,A 0.000,B 0.000,C 90.000,E1 161.873} C_DIS
LIN {X 0.054,Y -606.374,Z 1093.692,A 0.000,B 0.000,C 90.000,E1 160.550} C_DIS
LIN {X -0.123,Y -610.338,Z 1093.685,A 0.000,B 0.000,C 90.000,E1 159.263} C_DIS
LIN {X -0.192,Y -613.411,Z 1093.679,A 0.000,B 0.000,C 90.000,E1 158.230} C_DIS
LIN {X 0.002,Y -616.297,Z 1093.673,A 0.000,B 0.000,C 90.000,E1 157.177} C_DIS
LIN {X -0.332,Y -619.173,Z 1093.667,A 0.000,B 0.000,C 90.000,E1 156.177} C_DIS
LIN {X 0.192,Y -622.490,Z 1093.660,A 0.000,B 0.000,C 90.000,E1 154.845} C_DIS
LIN {X -0.059,Y -625.738,Z 1093.653,A 0.000,B 0.000,C 90.000,E1 153.589} C_DIS
LIN {X -0.005,Y -628.164,Z 1093.648,A 0.000,B 0.000,C 90.000,E1 152.564} C_DIS
LIN {X -0.125,Y -631.698,Z 1093.639,A 0.000,B 0.000,C 90.000,E1 151.051} C_DIS
LIN {X -0.202,Y -634.428,Z 1093.632,A 0.000,B 0.000,C 90.000,E1 149.793} C_DIS
LIN {X -0.236,Y -637.133,Z 1093.625,A 0.000,B 0.000,C 90.000,E1 148.535} C_DIS
LIN {X 0.146,Y -640.209,Z 1093.617,A 0.000,B 0.000,C 90.000,E1 146.993} C_DIS
LIN {X -0.129,Y -643.073,Z 1093.608,A 0.000,B 0.000,C 90.000,E1 145.515} C_DIS
LIN {X -0.292,Y -646.359,Z 1093.599,A 0.000,B 0.000,C 90.000,E1 143.783} C_DIS
LIN {X -0.138,Y -649.568,Z 1093.589,A 0.000,B 0.000,C 90.000,E1 142.029} C_DIS
LIN {X 0.104,Y -652.852,Z 1093.579,A 0.000,B 0.000,C 90.000,E1 140.275} C_DIS
LIN {X -0.028,Y -654.749,Z 1093.574,A 0.000,B 0.000,C 90.000,E1 139.299} C_DIS
LIN {X -0.175,Y -657.214,Z 1093.567,A 0.000,B 0.000,C 90.000,E1 138.081} C_DIS
LIN {X 0.138,Y -660.254,Z 1093.559,A 0.000,B 0.000,C 90.000,E1 136.581} C_DIS
LIN {X 0.017,Y -666.312,Z 1093.544,A 0.000,B 0.000,C 90.000,E1 133.905} C_DIS
LIN {X 0.031,Y -669.952,Z 1093.536,A 0.000,B 0.000,C 90.000,E1 132.447} C_DIS
LIN {X -0.267,Y -674.851,Z 1093.525,A 0.000,B 0.000,C 90.000,E1 130.539} C_DIS
LIN {X -0.336,Y -680.245,Z 1093.513,A 0.000,B 0.000,C 90.000,E1 128.382} C_DIS
LIN {X -0.358,Y -683.999,Z 1093.505,A 0.000,B 0.000,C 90.000,E1 126.950} C_DIS
LIN {X 0.040,Y -686.397,Z 1093.500,A 0.000,B 0.000,C 90.000,E1 125.964} C_DIS
LIN {X -0.090,Y -688.719,Z 1093.495,A 0.000,B 0.000,C 90.000,E1 125.025} C_DIS
LIN {X -0.140,Y -692.760,Z 1093.485,A 0.000,B 0.000,C 90.000,E1 123.372} C_DIS
LIN {X -0.015,Y -695.065,Z 1093.480,A 0.000,B 0.000,C 90.000,E1 122.418} C_DIS
LIN {X -0.208,Y -697.834,Z 1093.474,A 0.000,B 0.000,C 90.000,E1 121.258} C_DIS
LIN {X -0.385,Y -699.731,Z 1093.468,A 0.000,B 0.000,C 90.000,E1 120.335} C_DIS
LIN {X 0.076,Y -701.382,Z 1093.463,A 0.000,B 0.000,C 90.000,E1 119.361} C_DIS
LIN {X -0.049,Y -702.641,Z 1093.458,A 0.000,B 0.000,C 90.000,E1 118.437} C_DIS
LIN {X 0.172,Y -703.373,Z 1093.454,A 0.000,B 0.000,C 90.000,E1 117.719} C_DIS
LIN {X 0.025,Y -704.285,Z 1093.448,A 0.000,B 0.000,C 90.000,E1 116.565} C_DIS
LIN {X -0.094,Y -705.102,Z 1093.443,A 0.000,B 0.000,C 90.000,E1 115.643} C_DIS
LIN {X 0.180,Y -705.387,Z 1093.440,A 0.000,B 0.000,C 90.000,E1 115.155} C_DIS
LIN {X -0.177,Y -705.404,Z 1093.437,A 0.000,B 0.000,C 90.000,E1 114.719} C_DIS
LIN {X 0.113,Y -705.229,Z 1093.436,A 0.000,B 0.000,C 90.000,E1 114.463} C_DIS
LIN {X -0.243,Y -704.599,Z 1093.433,A 0.000,B 0.000,C 90.000,E1 114.027} C_DIS
LIN {X 0.326,Y -702.951,Z 1093.431,A 0.000,B 0.000,C 90.000,E1 113.515} C_DIS
LIN {X -0.318,Y -701.965,Z 1093.430,A 0.000,B 0.000,C 90.000,E1 113.334} C_DIS
LIN {X 0.226,Y -698.221,Z 1093.427,A 0.000,B 0.000,C 90.000,E1 112.823} C_DIS
LIN {X 0.086,Y -697.185,Z 1093.426,A 0.000,B 0.000,C 90.000,E1 112.717} C_DIS
LIN {X 0.217,Y -695.681,Z 1093.426,A 0.000,B 0.000,C 90.000,E1 112.589} C_DIS
LIN {X -0.140,Y -693.552,Z 1093.425,A 0.000,B 0.000,C 90.000,E1 112.514} C_DIS
LIN {X -0.238,Y -686.101,Z 1093.423,A 0.000,B 0.000,C 90.000,E1 112.206} C_DIS
LIN {X -0.030,Y -684.777,Z 1093.423,A 0.000,B 0.000,C 90.000,E1 112.153} C_DIS
LIN {X 0.090,Y -675.938,Z 1093.422,A 0.000,B 0.000,C 90.000,E1 112.025} C_DIS
LIN {X 0.033,Y -604.545,Z 1093.422,A 0.000,B 0.000,C 90.000,E1 112.025} C_DIS
LIN {X 0.066,Y -601.010,Z 1093.421,A 0.000,B 0.000,C 90.000,E1 111.844} C_DIS
LIN {X -0.126,Y -595.225,Z 1093.419,A 0.000,B 0.000,C 90.000,E1 111.461} C_DIS
LIN {X -0.126,Y -587.109,Z 1093.416,A 0.000,B 0.000,C 90.000,E1 110.791} C_DIS
LIN {X 0.164,Y -576.028,Z 1093.410,A 0.000,B 0.000,C 90.000,E1 109.812} C_DIS
LIN {X 0.160,Y -572.971,Z 1093.409,A 0.000,B 0.000,C 90.000,E1 109.577} C_DIS
LIN {X -0.087,Y -568.424,Z 1093.407,A 0.000,B 0.000,C 90.000,E1 109.268} C_DIS
LIN {X 0.246,Y -560.125,Z 1093.404,A 0.000,B 0.000,C 90.000,E1 108.725} C_DIS
LIN {X 0.128,Y -553.763,Z 1093.402,A 0.000,B 0.000,C 90.000,E1 108.362} C_DIS
LIN {X 0.133,Y -549.558,Z 1093.400,A 0.000,B 0.000,C 90.000,E1 108.055} C_DIS
LIN {X 0.124,Y -548.262,Z 1093.399,A 0.000,B 0.000,C 90.000,E1 107.873} C_DIS
LIN {X 0.082,Y -548.243,Z 1093.399,A 0.000,B 0.000,C 90.000,E1 107.873} C_DIS
LIN {X 0.203,Y -547.863,Z 1093.397,A 0.000,B 0.000,C 90.000,E1 107.457} C_DIS
LIN {X 0.132,Y -547.948,Z 1093.395,A 0.000,B 0.000,C 90.000,E1 106.985} C_DIS
LIN {X 0.193,Y -548.549,Z 1093.390,A 0.000,B 0.000,C 90.000,E1 106.134} C_DIS
LIN {X 0.114,Y -549.896,Z 1093.379,A 0.000,B 0.000,C 90.000,E1 104.175} C_DIS
LIN {X -0.071,Y -551.722,Z 1093.366,A 0.000,B 0.000,C 90.000,E1 101.951} C_DIS
LIN {X -0.139,Y -552.803,Z 1093.360,A 0.000,B 0.000,C 90.000,E1 100.838} C_DIS
LIN {X 0.081,Y -554.842,Z 1093.349,A 0.000,B 0.000,C 90.000,E1 98.859} C_DIS
LIN {X 0.262,Y -556.940,Z 1093.339,A 0.000,B 0.000,C 90.000,E1 96.891} C_DIS
LIN {X 0.091,Y -558.150,Z 1093.332,A 0.000,B 0.000,C 90.000,E1 95.796} C_DIS
LIN {X 0.014,Y -559.417,Z 1093.325,A 0.000,B 0.000,C 90.000,E1 94.416} C_DIS
LIN {X -0.046,Y -560.375,Z 1093.317,A 0.000,B 0.000,C 90.000,E1 93.037} C_DIS
LIN {X -0.125,Y -561.117,Z 1093.309,A 0.000,B 0.000,C 90.000,E1 91.661} C_DIS
LIN {X 0.261,Y -561.701,Z 1093.303,A 0.000,B 0.000,C 90.000,E1 90.516} C_DIS
LIN {X -0.263,Y -562.462,Z 1093.294,A 0.000,B 0.000,C 90.000,E1 88.912} C_DIS
LIN {X 0.260,Y -563.075,Z 1093.286,A 0.000,B 0.000,C 90.000,E1 87.478} C_DIS
LIN {X -0.193,Y -563.704,Z 1093.277,A 0.000,B 0.000,C 90.000,E1 85.869} C_DIS
LIN {X -0.168,Y -564.306,Z 1093.269,A 0.000,B 0.000,C 90.000,E1 84.489} C_DIS
LIN {X 0.104,Y -564.901,Z 1093.259,A 0.000,B 0.000,C 90.000,E1 82.534} C_DIS
LIN {X 0.278,Y -565.388,Z 1093.251,A 0.000,B 0.000,C 90.000,E1 81.141} C_DIS
LIN {X 0.255,Y -566.160,Z 1093.240,A 0.000,B 0.000,C 90.000,E1 79.218} C_DIS
LIN {X 0.068,Y -566.904,Z 1093.231,A 0.000,B 0.000,C 90.000,E1 77.589} C_DIS
LIN {X -0.240,Y -567.937,Z 1093.220,A 0.000,B 0.000,C 90.000,E1 75.700} C_DIS
LIN {X 0.005,Y -568.948,Z 1093.211,A 0.000,B 0.000,C 90.000,E1 74.031} C_DIS
LIN {X -0.104,Y -570.383,Z 1093.201,A 0.000,B 0.000,C 90.000,E1 72.127} C_DIS
LIN {X 0.164,Y -571.997,Z 1093.190,A 0.000,B 0.000,C 90.000,E1 70.188} C_DIS
LIN {X -0.057,Y -573.264,Z 1093.182,A 0.000,B 0.000,C 90.000,E1 68.847} C_DIS
LIN {X 0.154,Y -574.866,Z 1093.172,A 0.000,B 0.000,C 90.000,E1 66.922} C_DIS
LIN {X 0.030,Y -576.156,Z 1093.163,A 0.000,B 0.000,C 90.000,E1 65.305} C_DIS
LIN {X 0.267,Y -577.481,Z 1093.152,A 0.000,B 0.000,C 90.000,E1 63.384} C_DIS
LIN {X 0.318,Y -578.342,Z 1093.145,A 0.000,B 0.000,C 90.000,E1 62.025} C_DIS
LIN {X -0.270,Y -579.371,Z 1093.136,A 0.000,B 0.000,C 90.000,E1 60.461} C_DIS
LIN {X 0.095,Y -580.379,Z 1093.125,A 0.000,B 0.000,C 90.000,E1 58.535} C_DIS
LIN {X -0.034,Y -581.110,Z 1093.118,A 0.000,B 0.000,C 90.000,E1 57.199} C_DIS
LIN {X -0.157,Y -581.908,Z 1093.109,A 0.000,B 0.000,C 90.000,E1 55.595} C_DIS
LIN {X -0.256,Y -582.568,Z 1093.100,A 0.000,B 0.000,C 90.000,E1 53.989} C_DIS
LIN {X 0.276,Y -582.857,Z 1093.095,A 0.000,B 0.000,C 90.000,E1 53.130} C_DIS
LIN {X -0.108,Y -583.183,Z 1093.088,A 0.000,B 0.000,C 90.000,E1 51.823} C_DIS
LIN {X 0.058,Y -583.153,Z 1093.079,A 0.000,B 0.000,C 90.000,E1 50.194} C_DIS
LIN {X 0.042,Y -582.869,Z 1093.071,A 0.000,B 0.000,C 90.000,E1 48.852} C_DIS
LIN {X 0.134,Y -582.254,Z 1093.063,A 0.000,B 0.000,C 90.000,E1 47.229} C_DIS
LIN {X 0.052,Y -581.655,Z 1093.055,A 0.000,B 0.000,C 90.000,E1 45.891} C_DIS
LIN {X -0.190,Y -580.950,Z 1093.049,A 0.000,B 0.000,C 90.000,E1 44.838} C_DIS
LIN {X -0.173,Y -580.265,Z 1093.045,A 0.000,B 0.000,C 90.000,E1 44.028} C_DIS
LIN {X -0.292,Y -578.797,Z 1093.037,A 0.000,B 0.000,C 90.000,E1 42.690} C_DIS
LIN {X -0.161,Y -577.370,Z 1093.031,A 0.000,B 0.000,C 90.000,E1 41.595} C_DIS
LIN {X -0.144,Y -576.126,Z 1093.026,A 0.000,B 0.000,C 90.000,E1 40.782} C_DIS
LIN {X -0.063,Y -574.328,Z 1093.021,A 0.000,B 0.000,C 90.000,E1 39.688} C_DIS
LIN {X 0.197,Y -571.639,Z 1093.013,A 0.000,B 0.000,C 90.000,E1 38.302} C_DIS
LIN {X -0.198,Y -569.668,Z 1093.008,A 0.000,B 0.000,C 90.000,E1 37.523} C_DIS
LIN {X 0.064,Y -568.304,Z 1093.005,A 0.000,B 0.000,C 90.000,E1 36.950} C_DIS
LIN {X -0.022,Y -565.837,Z 1093.001,A 0.000,B 0.000,C 90.000,E1 36.137} C_DIS
LIN {X -0.012,Y -563.037,Z 1092.996,A 0.000,B 0.000,C 90.000,E1 35.311} C_DIS
LIN {X 0.094,Y -562.110,Z 1092.995,A 0.000,B 0.000,C 90.000,E1 35.025} C_DIS
LIN {X 0.071,Y -558.791,Z 1092.990,A 0.000,B 0.000,C 90.000,E1 34.199} C_DIS
LIN {X 0.014,Y -555.109,Z 1092.985,A 0.000,B 0.000,C 90.000,E1 33.372} C_DIS
LIN {X -0.088,Y -551.146,Z 1092.981,A 0.000,B 0.000,C 90.000,E1 32.546} C_DIS
LIN {X 0.353,Y -547.549,Z 1092.977,A 0.000,B 0.000,C 90.000,E1 31.799} C_DIS
LIN {X 0.030,Y -542.287,Z 1092.971,A 0.000,B 0.000,C 90.000,E1 30.846} C_DIS
LIN {X 0.104,Y -538.116,Z 1092.968,A 0.000,B 0.000,C 90.000,E1 30.129} C_DIS
LIN {X 0.146,Y -533.683,Z 1092.964,A 0.000,B 0.000,C 90.000,E1 29.411} C_DIS
LIN {X -0.024,Y -530.871,Z 1092.961,A 0.000,B 0.000,C 90.000,E1 28.999} C_DIS
LIN {X -0.149,Y -526.862,Z 1092.958,A 0.000,B 0.000,C 90.000,E1 28.437} C_DIS
LIN {X 0.109,Y -523.737,Z 1092.956,A 0.000,B 0.000,C 90.000,E1 27.975} C_DIS
LIN {X 0.165,Y -518.181,Z 1092.952,A 0.000,B 0.000,C 90.000,E1 27.257} C_DIS
LIN {X -0.037,Y -513.314,Z 1092.948,A 0.000,B 0.000,C 90.000,E1 26.693} C_DIS
LIN {X -0.267,Y -505.424,Z 1092.943,A 0.000,B 0.000,C 90.000,E1 25.848} C_DIS
LIN {X -0.325,Y -500.056,Z 1092.940,A 0.000,B 0.000,C 90.000,E1 25.283} C_DIS
LIN {X -0.039,Y -490.373,Z 1092.935,A 0.000,B 0.000,C 90.000,E1 24.259} C_DIS
LIN {X 0.013,Y -478.696,Z 1092.929,A 0.000,B 0.000,C 90.000,E1 23.153} C_DIS
LIN {X -0.021,Y -473.005,Z 1092.926,A 0.000,B 0.000,C 90.000,E1 22.642} C_DIS
LIN {X -0.111,Y -461.415,Z 1092.920,A 0.000,B 0.000,C 90.000,E1 21.642} C_DIS
LIN {X -0.023,Y -444.975,Z 1092.912,A 0.000,B 0.000,C 90.000,E1 20.174} C_DIS
LIN {X -0.117,Y -431.903,Z 1092.905,A 0.000,B 0.000,C 90.000,E1 18.960} C_DIS
LIN {X 0.004,Y -419.303,Z 1092.898,A 0.000,B 0.000,C 90.000,E1 17.638} C_DIS
LIN {X -0.003,Y -407.019,Z 1092.890,A 0.000,B 0.000,C 90.000,E1 16.205} C_DIS
LIN {X 0.009,Y -399.308,Z 1092.884,A 0.000,B 0.000,C 90.000,E1 15.190} C_DIS
LIN {X 0.016,Y -397.434,Z 1092.883,A 0.000,B 0.000,C 90.000,E1 14.898} C_DIS
LIN {X -0.063,Y -395.627,Z 1092.881,A 0.000,B 0.000,C 90.000,E1 14.592} C_DIS
LIN {X 0.134,Y -393.495,Z 1092.878,A 0.000,B 0.000,C 90.000,E1 14.064} C_DIS
LIN {X 0.116,Y -392.380,Z 1092.875,A 0.000,B 0.000,C 90.000,E1 13.536} C_DIS
LIN {X 0.160,Y -392.139,Z 1092.873,A 0.000,B 0.000,C 90.000,E1 13.175} C_DIS
LIN {X 0.111,Y -392.063,Z 1092.871,A 0.000,B 0.000,C 90.000,E1 12.827} C_DIS
LIN {X 0.133,Y -392.570,Z 1092.867,A 0.000,B 0.000,C 90.000,E1 12.119} C_DIS
LIN {X 0.001,Y -394.042,Z 1092.862,A 0.000,B 0.000,C 90.000,E1 11.074} C_DIS
LIN {X 0.197,Y -400.251,Z 1092.844,A 0.000,B 0.000,C 90.000,E1 7.871} C_DIS
LIN {X -0.001,Y -405.934,Z 1092.830,A 0.000,B 0.000,C 90.000,E1 5.454} C_DIS
LIN {X 0.000,Y -406.770,Z 1092.828,A 0.000,B 0.000,C 90.000,E1 5.106} C_DIS
LIN {X -0.024,Y -409.188,Z 1092.825,A 0.000,B 0.000,C 90.000,E1 4.416} C_DIS
LIN {X -0.019,Y -412.073,Z 1092.822,A 0.000,B 0.000,C 90.000,E1 3.898} C_DIS
LIN {X -0.025,Y -413.470,Z 1092.821,A 0.000,B 0.000,C 90.000,E1 3.726} C_DIS
LIN {X 0.195,Y -417.226,Z 1092.819,A 0.000,B 0.000,C 90.000,E1 3.326} C_DIS
LIN {X -0.051,Y -424.233,Z 1092.816,A 0.000,B 0.000,C 90.000,E1 2.865} C_DIS
LIN {X 0.172,Y -434.073,Z 1092.812,A 0.000,B 0.000,C 90.000,E1 2.178} C_DIS
LIN {X 0.223,Y -450.577,Z 1092.806,A 0.000,B 0.000,C 90.000,E1 1.088} C_DIS
LIN {X 0.089,Y -470.011,Z 1092.799,A 0.000,B 0.000,C 90.000,E1 359.885} C_DIS
LIN {X 0.203,Y -479.815,Z 1092.796,A 0.000,B 0.000,C 90.000,E1 359.255} C_DIS
LIN {X 0.234,Y -489.501,Z 1092.793,A 0.000,B 0.000,C 90.000,E1 358.625} C_DIS
LIN {X 0.111,Y -498.901,Z 1092.789,A 0.000,B 0.000,C 90.000,E1 357.993} C_DIS
LIN {X 0.248,Y -505.045,Z 1092.786,A 0.000,B 0.000,C 90.000,E1 357.535} C_DIS
LIN {X -0.245,Y -509.637,Z 1092.785,A 0.000,B 0.000,C 90.000,E1 357.249} C_DIS
LIN {X 0.113,Y -516.865,Z 1092.781,A 0.000,B 0.000,C 90.000,E1 356.617} C_DIS
LIN {X -0.251,Y -523.826,Z 1092.778,A 0.000,B 0.000,C 90.000,E1 356.045} C_DIS
LIN {X -0.118,Y -527.930,Z 1092.776,A 0.000,B 0.000,C 90.000,E1 355.641} C_DIS
LIN {X -0.147,Y -534.098,Z 1092.772,A 0.000,B 0.000,C 90.000,E1 355.008} C_DIS
LIN {X -0.177,Y -540.048,Z 1092.768,A 0.000,B 0.000,C 90.000,E1 354.318} C_DIS
LIN {X 0.247,Y -545.581,Z 1092.765,A 0.000,B 0.000,C 90.000,E1 353.571} C_DIS
LIN {X -0.192,Y -549.704,Z 1092.761,A 0.000,B 0.000,C 90.000,E1 353.053} C_DIS
LIN {X -0.241,Y -554.224,Z 1092.757,A 0.000,B 0.000,C 90.000,E1 352.356} C_DIS
LIN {X -0.075,Y -557.575,Z 1092.754,A 0.000,B 0.000,C 90.000,E1 351.781} C_DIS
LIN {X -0.052,Y -561.254,Z 1092.750,A 0.000,B 0.000,C 90.000,E1 351.084} C_DIS
LIN {X 0.253,Y -564.010,Z 1092.747,A 0.000,B 0.000,C 90.000,E1 350.500} C_DIS
LIN {X 0.273,Y -568.879,Z 1092.741,A 0.000,B 0.000,C 90.000,E1 349.398} C_DIS
LIN {X -0.103,Y -573.268,Z 1092.735,A 0.000,B 0.000,C 90.000,E1 348.342} C_DIS
LIN {X -0.208,Y -578.236,Z 1092.728,A 0.000,B 0.000,C 90.000,E1 346.992} C_DIS
LIN {X -0.236,Y -582.813,Z 1092.720,A 0.000,B 0.000,C 90.000,E1 345.644} C_DIS
LIN {X -0.288,Y -586.284,Z 1092.714,A 0.000,B 0.000,C 90.000,E1 344.574} C_DIS
LIN {X -0.291,Y -589.577,Z 1092.708,A 0.000,B 0.000,C 90.000,E1 343.504} C_DIS
LIN {X 0.052,Y -594.344,Z 1092.699,A 0.000,B 0.000,C 90.000,E1 341.873} C_DIS
LIN {X 0.342,Y -597.300,Z 1092.693,A 0.000,B 0.000,C 90.000,E1 340.786} C_DIS
LIN {X -0.192,Y -600.474,Z 1092.686,A 0.000,B 0.000,C 90.000,E1 339.518} C_DIS
LIN {X -0.100,Y -602.243,Z 1092.682,A 0.000,B 0.000,C 90.000,E1 338.720} C_DIS
LIN {X -0.060,Y -604.317,Z 1092.676,A 0.000,B 0.000,C 90.000,E1 337.667} C_DIS
LIN {X 0.069,Y -605.710,Z 1092.672,A 0.000,B 0.000,C 90.000,E1 336.869} C_DIS
LIN {X -0.104,Y -606.937,Z 1092.667,A 0.000,B 0.000,C 90.000,E1 336.102} C_DIS
LIN {X -0.053,Y -608.711,Z 1092.660,A 0.000,B 0.000,C 90.000,E1 334.793} C_DIS
LIN {X -0.269,Y -610.151,Z 1092.653,A 0.000,B 0.000,C 90.000,E1 333.512} C_DIS
LIN {X 0.117,Y -610.932,Z 1092.647,A 0.000,B 0.000,C 90.000,E1 332.436} C_DIS
LIN {X 0.290,Y -611.463,Z 1092.643,A 0.000,B 0.000,C 90.000,E1 331.641} C_DIS
LIN {X -0.092,Y -611.842,Z 1092.637,A 0.000,B 0.000,C 90.000,E1 330.639} C_DIS
LIN {X -0.164,Y -611.899,Z 1092.634,A 0.000,B 0.000,C 90.000,E1 330.127} C_DIS
LIN {X -0.012,Y -611.520,Z 1092.628,A 0.000,B 0.000,C 90.000,E1 329.076} C_DIS
LIN {X -0.072,Y -610.699,Z 1092.622,A 0.000,B 0.000,C 90.000,E1 328.043} C_DIS
LIN {X 0.047,Y -609.425,Z 1092.617,A 0.000,B 0.000,C 90.000,E1 326.993} C_DIS
LIN {X -0.040,Y -607.614,Z 1092.611,A 0.000,B 0.000,C 90.000,E1 325.960} C_DIS
LIN {X 0.110,Y -605.210,Z 1092.604,A 0.000,B 0.000,C 90.000,E1 324.642} C_DIS
LIN {X 0.341,Y -602.420,Z 1092.595,A 0.000,B 0.000,C 90.000,E1 323.050} C_DIS
LIN {X -0.076,Y -599.119,Z 1092.585,A 0.000,B 0.000,C 90.000,E1 321.251} C_DIS
LIN {X -0.054,Y -597.140,Z 1092.579,A 0.000,B 0.000,C 90.000,E1 320.194} C_DIS
LIN {X 0.169,Y -594.948,Z 1092.572,A 0.000,B 0.000,C 90.000,E1 318.852} C_DIS
LIN {X 0.131,Y -592.918,Z 1092.566,A 0.000,B 0.000,C 90.000,E1 317.796} C_DIS
LIN {X 0.266,Y -591.245,Z 1092.561,A 0.000,B 0.000,C 90.000,E1 316.986} C_DIS
LIN {X -0.259,Y -588.575,Z 1092.555,A 0.000,B 0.000,C 90.000,E1 315.972} C_DIS
LIN {X -0.162,Y -586.335,Z 1092.551,A 0.000,B 0.000,C 90.000,E1 315.162} C_DIS
LIN {X 0.165,Y -585.018,Z 1092.548,A 0.000,B 0.000,C 90.000,E1 314.595} C_DIS
LIN {X 0.120,Y -581.121,Z 1092.540,A 0.000,B 0.000,C 90.000,E1 313.257} C_DIS
LIN {X -0.272,Y -576.334,Z 1092.531,A 0.000,B 0.000,C 90.000,E1 311.676} C_DIS
LIN {X 0.023,Y -574.366,Z 1092.528,A 0.000,B 0.000,C 90.000,E1 311.105} C_DIS
LIN {X 0.248,Y -572.205,Z 1092.525,A 0.000,B 0.000,C 90.000,E1 310.539} C_DIS
LIN {X -0.036,Y -569.164,Z 1092.522,A 0.000,B 0.000,C 90.000,E1 309.886} C_DIS
LIN {X -0.104,Y -565.109,Z 1092.517,A 0.000,B 0.000,C 90.000,E1 309.072} C_DIS
LIN {X -0.216,Y -560.895,Z 1092.512,A 0.000,B 0.000,C 90.000,E1 308.257} C_DIS
LIN {X 0.194,Y -556.981,Z 1092.509,A 0.000,B 0.000,C 90.000,E1 307.523} C_DIS
LIN {X -0.015,Y -552.071,Z 1092.504,A 0.000,B 0.000,C 90.000,E1 306.710} C_DIS
LIN {X 0.050,Y -550.241,Z 1092.502,A 0.000,B 0.000,C 90.000,E1 306.423} C_DIS
LIN {X -0.026,Y -547.802,Z 1092.500,A 0.000,B 0.000,C 90.000,E1 306.011} C_DIS
LIN {X -0.159,Y -546.936,Z 1092.499,A 0.000,B 0.000,C 90.000,E1 305.884} C_DIS
LIN {X -0.069,Y -544.246,Z 1092.496,A 0.000,B 0.000,C 90.000,E1 305.311} C_DIS
LIN {X -0.033,Y -543.238,Z 1092.495,A 0.000,B 0.000,C 90.000,E1 305.025} C_DIS
LIN {X -0.141,Y -541.424,Z 1092.492,A 0.000,B 0.000,C 90.000,E1 304.612} C_DIS
LIN {X 0.025,Y -541.169,Z 1092.491,A 0.000,B 0.000,C 90.000,E1 304.452} C_DIS
LIN {X -0.259,Y -540.262,Z 1092.490,A 0.000,B 0.000,C 90.000,E1 304.199} C_DIS
LIN {X -0.237,Y -539.259,Z 1092.488,A 0.000,B 0.000,C 90.000,E1 303.913} C_DIS
LIN {X 0.312,Y -537.731,Z 1092.484,A 0.000,B 0.000,C 90.000,E1 303.086} C_DIS
LIN {X 0.027,Y -537.457,Z 1092.482,A 0.000,B 0.000,C 90.000,E1 302.832} C_DIS
LIN {X -0.081,Y -536.917,Z 1092.474,A 0.000,B 0.000,C 90.000,E1 301.416} C_DIS
LIN {X 0.081,Y -537.139,Z 1092.468,A 0.000,B 0.000,C 90.000,E1 300.256} C_DIS
LIN {X 0.063,Y -537.674,Z 1092.455,A 0.000,B 0.000,C 90.000,E1 297.975} C_DIS
LIN {X 0.087,Y -538.628,Z 1092.444,A 0.000,B 0.000,C 90.000,E1 295.976} C_DIS
LIN {X -0.018,Y -539.096,Z 1092.438,A 0.000,B 0.000,C 90.000,E1 294.847} C_DIS
LIN {X 0.108,Y -539.470,Z 1092.432,A 0.000,B 0.000,C 90.000,E1 293.695} C_DIS
LIN {X -0.017,Y -540.052,Z 1092.421,A 0.000,B 0.000,C 90.000,E1 291.716} C_DIS
LIN {X -0.081,Y -540.357,Z 1092.413,A 0.000,B 0.000,C 90.000,E1 290.301} C_DIS
LIN {X 0.183,Y -540.370,Z 1092.405,A 0.000,B 0.000,C 90.000,E1 288.852} C_DIS
LIN {X 0.174,Y -540.275,Z 1092.400,A 0.000,B 0.000,C 90.000,E1 288.000} C_DIS
LIN {X -0.241,Y -540.034,Z 1092.392,A 0.000,B 0.000,C 90.000,E1 286.622} C_DIS
LIN {X -0.206,Y -539.686,Z 1092.386,A 0.000,B 0.000,C 90.000,E1 285.481} C_DIS
LIN {X -0.259,Y -539.145,Z 1092.378,A 0.000,B 0.000,C 90.000,E1 284.064} C_DIS
LIN {X 0.202,Y -538.501,Z 1092.370,A 0.000,B 0.000,C 90.000,E1 282.591} C_DIS
LIN {X 0.010,Y -537.799,Z 1092.362,A 0.000,B 0.000,C 90.000,E1 281.186} C_DIS
LIN {X -0.171,Y -536.809,Z 1092.351,A 0.000,B 0.000,C 90.000,E1 279.208} C_DIS
LIN {X 0.036,Y -536.049,Z 1092.343,A 0.000,B 0.000,C 90.000,E1 277.757} C_DIS
LIN {X 0.142,Y -535.231,Z 1092.334,A 0.000,B 0.000,C 90.000,E1 276.030} C_DIS
LIN {X 0.209,Y -534.669,Z 1092.327,A 0.000,B 0.000,C 90.000,E1 274.878} C_DIS
LIN {X 0.268,Y -533.692,Z 1092.316,A 0.000,B 0.000,C 90.000,E1 272.865} C_DIS
LIN {X 0.236,Y -532.660,Z 1092.303,A 0.000,B 0.000,C 90.000,E1 270.573} C_DIS
LIN {X 0.186,Y -531.751,Z 1092.294,A 0.000,B 0.000,C 90.000,E1 268.854} C_DIS
LIN {X 0.124,Y -530.732,Z 1092.284,A 0.000,B 0.000,C 90.000,E1 267.135} C_DIS
LIN {X 0.097,Y -530.245,Z 1092.279,A 0.000,B 0.000,C 90.000,E1 266.274} C_DIS
LIN {X 0.084,Y -529.535,Z 1092.273,A 0.000,B 0.000,C 90.000,E1 265.122} C_DIS
LIN {X 0.066,Y -528.692,Z 1092.267,A 0.000,B 0.000,C 90.000,E1 263.970} C_DIS
LIN {X 0.012,Y -527.949,Z 1092.262,A 0.000,B 0.000,C 90.000,E1 263.109} C_DIS
LIN {X 0.012,Y -525.793,Z 1092.250,A 0.000,B 0.000,C 90.000,E1 261.084} C_DIS
LIN {X 0.064,Y -523.117,Z 1092.236,A 0.000,B 0.000,C 90.000,E1 258.465} C_DIS
LIN {X 0.228,Y -521.097,Z 1092.225,A 0.000,B 0.000,C 90.000,E1 256.408} C_DIS
LIN {X -0.028,Y -519.434,Z 1092.215,A 0.000,B 0.000,C 90.000,E1 254.685} C_DIS
LIN {X 0.306,Y -517.261,Z 1092.204,A 0.000,B 0.000,C 90.000,E1 252.598} C_DIS
LIN {X 0.107,Y -515.336,Z 1092.194,A 0.000,B 0.000,C 90.000,E1 250.859} C_DIS
LIN {X 0.077,Y -513.717,Z 1092.186,A 0.000,B 0.000,C 90.000,E1 249.390} C_DIS
LIN {X 0.018,Y -511.961,Z 1092.177,A 0.000,B 0.000,C 90.000,E1 247.922} C_DIS
LIN {X 0.111,Y -510.084,Z 1092.169,A 0.000,B 0.000,C 90.000,E1 246.433} C_DIS
LIN {X 0.274,Y -508.299,Z 1092.163,A 0.000,B 0.000,C 90.000,E1 245.229} C_DIS
LIN {X 0.046,Y -505.892,Z 1092.154,A 0.000,B 0.000,C 90.000,E1 243.768} C_DIS
LIN {X 0.072,Y -502.966,Z 1092.144,A 0.000,B 0.000,C 90.000,E1 241.975} C_DIS
LIN {X 0.210,Y -500.419,Z 1092.136,A 0.000,B 0.000,C 90.000,E1 240.461} C_DIS
LIN {X 0.156,Y -497.333,Z 1092.126,A 0.000,B 0.000,C 90.000,E1 238.663} C_DIS
LIN {X 0.166,Y -495.146,Z 1092.119,A 0.000,B 0.000,C 90.000,E1 237.454} C_DIS
LIN {X -0.166,Y -491.731,Z 1092.109,A 0.000,B 0.000,C 90.000,E1 235.674} C_DIS
LIN {X 0.303,Y -489.410,Z 1092.103,A 0.000,B 0.000,C 90.000,E1 234.402} C_DIS
LIN {X -0.113,Y -486.432,Z 1092.094,A 0.000,B 0.000,C 90.000,E1 232.924} C_DIS
LIN {X -0.117,Y -483.957,Z 1092.087,A 0.000,B 0.000,C 90.000,E1 231.698} C_DIS
LIN {X -0.049,Y -480.796,Z 1092.079,A 0.000,B 0.000,C 90.000,E1 230.150} C_DIS
LIN {X 0.019,Y -476.967,Z 1092.068,A 0.000,B 0.000,C 90.000,E1 228.286} C_DIS
LIN {X -0.025,Y -471.596,Z 1092.053,A 0.000,B 0.000,C 90.000,E1 225.486} C_DIS
LIN {X -0.174,Y -468.163,Z 1092.042,A 0.000,B 0.000,C 90.000,E1 223.623} C_DIS
LIN {X 0.209,Y -465.185,Z 1092.034,A 0.000,B 0.000,C 90.000,E1 222.000} C_DIS
LIN {X 0.020,Y -461.052,Z 1092.021,A 0.000,B 0.000,C 90.000,E1 219.806} C_DIS
LIN {X -0.047,Y -458.141,Z 1092.012,A 0.000,B 0.000,C 90.000,E1 218.222} C_DIS
LIN {X -0.012,Y -454.746,Z 1092.002,A 0.000,B 0.000,C 90.000,E1 216.297} C_DIS
LIN {X -0.119,Y -452.573,Z 1091.995,A 0.000,B 0.000,C 90.000,E1 215.025} C_DIS
LIN {X 0.110,Y -450.300,Z 1091.987,A 0.000,B 0.000,C 90.000,E1 213.706} C_DIS
LIN {X -0.023,Y -448.722,Z 1091.982,A 0.000,B 0.000,C 90.000,E1 212.752} C_DIS
LIN {X 0.103,Y -444.825,Z 1091.969,A 0.000,B 0.000,C 90.000,E1 210.463} C_DIS
LIN {X 0.067,Y -441.264,Z 1091.957,A 0.000,B 0.000,C 90.000,E1 208.180} C_DIS
LIN {X 0.009,Y -436.693,Z 1091.938,A 0.000,B 0.000,C 90.000,E1 204.899} C_DIS
LIN {X 0.083,Y -435.501,Z 1091.933,A 0.000,B 0.000,C 90.000,E1 203.898} C_DIS
LIN {X -0.028,Y -434.289,Z 1091.926,A 0.000,B 0.000,C 90.000,E1 202.589} C_DIS
LIN {X -0.035,Y -433.988,Z 1091.924,A 0.000,B 0.000,C 90.000,E1 202.259} C_DIS
LIN {X 0.066,Y -433.585,Z 1091.916,A 0.000,B 0.000,C 90.000,E1 200.918} C_DIS
LIN {X -0.059,Y -433.913,Z 1091.911,A 0.000,B 0.000,C 90.000,E1 199.939} C_DIS
LIN {X -0.005,Y -434.602,Z 1091.907,A 0.000,B 0.000,C 90.000,E1 199.268} C_DIS
LIN {X 0.051,Y -435.674,Z 1091.903,A 0.000,B 0.000,C 90.000,E1 198.598} C_DIS
LIN {X -0.023,Y -437.146,Z 1091.900,A 0.000,B 0.000,C 90.000,E1 197.946} C_DIS
LIN {X 0.051,Y -438.980,Z 1091.896,A 0.000,B 0.000,C 90.000,E1 197.275} C_DIS
LIN {X -0.159,Y -442.379,Z 1091.891,A 0.000,B 0.000,C 90.000,E1 196.315} C_DIS
LIN {X -0.140,Y -450.368,Z 1091.880,A 0.000,B 0.000,C 90.000,E1 194.356} C_DIS
LIN {X -0.199,Y -458.262,Z 1091.870,A 0.000,B 0.000,C 90.000,E1 192.591} C_DIS
LIN {X -0.106,Y -469.752,Z 1091.857,A 0.000,B 0.000,C 90.000,E1 190.197} C_DIS
LIN {X -0.066,Y -475.277,Z 1091.851,A 0.000,B 0.000,C 90.000,E1 189.095} C_DIS
LIN {X 0.079,Y -478.364,Z 1091.847,A 0.000,B 0.000,C 90.000,E1 188.454} C_DIS
LIN {X 0.271,Y -479.268,Z 1091.846,A 0.000,B 0.000,C 90.000,E1 188.276} C_DIS
LIN {X -0.104,Y -486.746,Z 1091.838,A 0.000,B 0.000,C 90.000,E1 186.777} C_DIS
LIN {X -0.056,Y -491.210,Z 1091.833,A 0.000,B 0.000,C 90.000,E1 185.853} C_DIS
LIN {X -0.115,Y -497.034,Z 1091.826,A 0.000,B 0.000,C 90.000,E1 184.645} C_DIS
LIN {X -0.215,Y -504.228,Z 1091.817,A 0.000,B 0.000,C 90.000,E1 183.151} C_DIS
LIN {X 0.212,Y -512.819,Z 1091.807,A 0.000,B 0.000,C 90.000,E1 181.318} C_DIS
LIN {X -0.143,Y -519.953,Z 1091.799,A 0.000,B 0.000,C 90.000,E1 179.885} C_DIS
LIN {X -0.130,Y -527.813,Z 1091.790,A 0.000,B 0.000,C 90.000,E1 178.282} C_DIS
LIN {X -0.189,Y -536.277,Z 1091.781,A 0.000,B 0.000,C 90.000,E1 176.560} C_DIS
LIN {X -0.058,Y -544.581,Z 1091.771,A 0.000,B 0.000,C 90.000,E1 174.837} C_DIS
LIN {X -0.094,Y -550.763,Z 1091.764,A 0.000,B 0.000,C 90.000,E1 173.571} C_DIS
LIN {X 0.033,Y -556.884,Z 1091.757,A 0.000,B 0.000,C 90.000,E1 172.299} C_DIS
LIN {X -0.046,Y -562.280,Z 1091.751,A 0.000,B 0.000,C 90.000,E1 171.197} C_DIS
LIN {X -0.050,Y -567.547,Z 1091.745,A 0.000,B 0.000,C 90.000,E1 170.095} C_DIS
LIN {X 0.207,Y -573.891,Z 1091.737,A 0.000,B 0.000,C 90.000,E1 168.701} C_DIS
LIN {X -0.209,Y -579.413,Z 1091.731,A 0.000,B 0.000,C 90.000,E1 167.521} C_DIS
LIN {X 0.130,Y -584.095,Z 1091.725,A 0.000,B 0.000,C 90.000,E1 166.408} C_DIS
LIN {X -0.217,Y -589.747,Z 1091.717,A 0.000,B 0.000,C 90.000,E1 165.102} C_DIS
LIN {X -0.165,Y -593.974,Z 1091.711,A 0.000,B 0.000,C 90.000,E1 164.031} C_DIS
LIN {X 0.220,Y -598.854,Z 1091.704,A 0.000,B 0.000,C 90.000,E1 162.670} C_DIS
LIN {X -0.001,Y -602.492,Z 1091.698,A 0.000,B 0.000,C 90.000,E1 161.638} C_DIS
LIN {X -0.168,Y -605.913,Z 1091.692,A 0.000,B 0.000,C 90.000,E1 160.604} C_DIS
LIN {X -0.051,Y -610.720,Z 1091.683,A 0.000,B 0.000,C 90.000,E1 159.028} C_DIS
LIN {X 0.107,Y -613.778,Z 1091.678,A 0.000,B 0.000,C 90.000,E1 157.975} C_DIS
LIN {X 0.001,Y -618.809,Z 1091.668,A 0.000,B 0.000,C 90.000,E1 156.177} C_DIS
LIN {X -0.307,Y -622.113,Z 1091.661,A 0.000,B 0.000,C 90.000,E1 154.921} C_DIS
LIN {X -0.294,Y -625.369,Z 1091.653,A 0.000,B 0.000,C 90.000,E1 153.640} C_DIS
LIN {X -0.242,Y -627.817,Z 1091.648,A 0.000,B 0.000,C 90.000,E1 152.615} C_DIS
LIN {X 0.191,Y -631.390,Z 1091.639,A 0.000,B 0.000,C 90.000,E1 151.051} C_DIS
LIN {X 0.110,Y -634.129,Z 1091.632,A 0.000,B 0.000,C 90.000,E1 149.793} C_DIS
LIN {X 0.071,Y -636.839,Z 1091.625,A 0.000,B 0.000,C 90.000,E1 148.535} C_DIS
LIN {X -0.046,Y -640.426,Z 1091.615,A 0.000,B 0.000,C 90.000,E1 146.786} C_DIS
LIN {X 0.213,Y -643.293,Z 1091.607,A 0.000,B 0.000,C 90.000,E1 145.261} C_DIS
LIN {X 0.002,Y -646.137,Z 1091.599,A 0.000,B 0.000,C 90.000,E1 143.783} C_DIS
LIN {X -0.322,Y -649.839,Z 1091.588,A 0.000,B 0.000,C 90.000,E1 141.823} C_DIS
LIN {X -0.138,Y -653.657,Z 1091.577,A 0.000,B 0.000,C 90.000,E1 139.828} C_DIS
LIN {X 0.075,Y -657.532,Z 1091.566,A 0.000,B 0.000,C 90.000,E1 137.838} C_DIS
LIN {X -0.056,Y -660.612,Z 1091.558,A 0.000,B 0.000,C 90.000,E1 136.377} C_DIS
LIN {X -0.187,Y -666.760,Z 1091.543,A 0.000,B 0.000,C 90.000,E1 133.704} C_DIS
LIN {X -0.136,Y -670.408,Z 1091.535,A 0.000,B 0.000,C 90.000,E1 132.243} C_DIS
LIN {X 0.024,Y -675.296,Z 1091.524,A 0.000,B 0.000,C 90.000,E1 130.297} C_DIS
LIN {X -0.062,Y -680.099,Z 1091.513,A 0.000,B 0.000,C 90.000,E1 128.382} C_DIS
LIN {X -0.086,Y -683.870,Z 1091.505,A 0.000,B 0.000,C 90.000,E1 126.950} C_DIS
LIN {X -0.244,Y -686.283,Z 1091.500,A 0.000,B 0.000,C 90.000,E1 126.011} C_DIS
LIN {X 0.180,Y -688.601,Z 1091.495,A 0.000,B 0.000,C 90.000,E1 125.025} C_DIS
LIN {X -0.089,Y -692.066,Z 1091.487,A 0.000,B 0.000,C 90.000,E1 123.627} C_DIS
LIN {X 0.254,Y -694.944,Z 1091.480,A 0.000,B 0.000,C 90.000,E1 122.418} C_DIS
LIN {X 0.060,Y -697.734,Z 1091.474,A 0.000,B 0.000,C 90.000,E1 121.258} C_DIS
LIN {X -0.117,Y -699.627,Z 1091.469,A 0.000,B 0.000,C 90.000,E1 120.335} C_DIS
LIN {X -0.267,Y -701.297,Z 1091.463,A 0.000,B 0.000,C 90.000,E1 119.411} C_DIS
LIN {X 0.217,Y -702.535,Z 1091.458,A 0.000,B 0.000,C 90.000,E1 118.437} C_DIS
LIN {X 0.097,Y -703.477,Z 1091.453,A 0.000,B 0.000,C 90.000,E1 117.513} C_DIS
LIN {X -0.136,Y -705.018,Z 1091.443,A 0.000,B 0.000,C 90.000,E1 115.668} C_DIS
LIN {X -0.195,Y -705.330,Z 1091.440,A 0.000,B 0.000,C 90.000,E1 115.207} C_DIS
LIN {X 0.085,Y -705.346,Z 1091.437,A 0.000,B 0.000,C 90.000,E1 114.719} C_DIS
LIN {X -0.267,Y -705.211,Z 1091.436,A 0.000,B 0.000,C 90.000,E1 114.515} C_DIS
LIN {X 0.018,Y -704.595,Z 1091.434,A 0.000,B 0.000,C 90.000,E1 114.027} C_DIS
LIN {X 0.305,Y -703.871,Z 1091.432,A 0.000,B 0.000,C 90.000,E1 113.770} C_DIS
LIN {X -0.056,Y -702.078,Z 1091.430,A 0.000,B 0.000,C 90.000,E1 113.334} C_DIS
LIN {X 0.219,Y -700.317,Z 1091.428,A 0.000,B 0.000,C 90.000,E1 113.078} C_DIS
LIN {X -0.242,Y -697.470,Z 1091.426,A 0.000,B 0.000,C 90.000,E1 112.770} C_DIS
LIN {X -0.111,Y -696.106,Z 1091.426,A 0.000,B 0.000,C 90.000,E1 112.642} C_DIS
LIN {X 0.111,Y -694.072,Z 1091.425,A 0.000,B 0.000,C 90.000,E1 112.514} C_DIS
LIN {X -0.051,Y -686.619,Z 1091.423,A 0.000,B 0.000,C 90.000,E1 112.206} C_DIS
LIN {X -0.268,Y -683.663,Z 1091.423,A 0.000,B 0.000,C 90.000,E1 112.153} C_DIS
LIN {X 0.056,Y -675.893,Z 1091.422,A 0.000,B 0.000,C 90.000,E1 112.025} C_DIS
LIN {X 0.002,Y -604.642,Z 1091.422,A 0.000,B 0.000,C 90.000,E1 112.025} C_DIS
LIN {X -0.108,Y -600.899,Z 1091.421,A 0.000,B 0.000,C 90.000,E1 111.844} C_DIS
LIN {X -0.017,Y -596.424,Z 1091.420,A 0.000,B 0.000,C 90.000,E1 111.535} C_DIS
LIN {X -0.269,Y -588.471,Z 1091.416,A 0.000,B 0.000,C 90.000,E1 110.918} C_DIS
LIN {X 0.195,Y -577.548,Z 1091.411,A 0.000,B 0.000,C 90.000,E1 109.939} C_DIS
LIN {X 0.171,Y -574.744,Z 1091.410,A 0.000,B 0.000,C 90.000,E1 109.704} C_DIS
LIN {X 0.102,Y -568.733,Z 1091.407,A 0.000,B 0.000,C 90.000,E1 109.268} C_DIS
LIN {X -0.108,Y -560.478,Z 1091.404,A 0.000,B 0.000,C 90.000,E1 108.779} C_DIS
LIN {X -0.218,Y -554.043,Z 1091.402,A 0.000,B 0.000,C 90.000,E1 108.417} C_DIS
LIN {X 0.313,Y -549.678,Z 1091.401,A 0.000,B 0.000,C 90.000,E1 108.055} C_DIS
LIN {X 0.071,Y -548.186,Z 1091.399,A 0.000,B 0.000,C 90.000,E1 107.873} C_DIS
LIN {X 0.029,Y -548.157,Z 1091.399,A 0.000,B 0.000,C 90.000,E1 107.873} C_DIS
LIN {X -0.195,Y -547.841,Z 1091.398,A 0.000,B 0.000,C 90.000,E1 107.638} C_DIS
LIN {X 0.144,Y -547.868,Z 1091.395,A 0.000,B 0.000,C 90.000,E1 107.040} C_DIS
LIN {X 0.296,Y -548.611,Z 1091.389,A 0.000,B 0.000,C 90.000,E1 105.898} C_DIS
LIN {X 0.087,Y -549.994,Z 1091.378,A 0.000,B 0.000,C 90.000,E1 103.953} C_DIS
LIN {X 0.039,Y -551.862,Z 1091.365,A 0.000,B 0.000,C 90.000,E1 101.715} C_DIS
LIN {X -0.029,Y -552.936,Z 1091.359,A 0.000,B 0.000,C 90.000,E1 100.602} C_DIS
LIN {X 0.065,Y -554.725,Z 1091.350,A 0.000,B 0.000,C 90.000,E1 98.916} C_DIS
LIN {X 0.240,Y -556.851,Z 1091.339,A 0.000,B 0.000,C 90.000,E1 96.947} C_DIS
LIN {X 0.066,Y -558.065,Z 1091.333,A 0.000,B 0.000,C 90.000,E1 95.853} C_DIS
LIN {X -0.014,Y -559.341,Z 1091.325,A 0.000,B 0.000,C 90.000,E1 94.473} C_DIS
LIN {X -0.075,Y -560.293,Z 1091.317,A 0.000,B 0.000,C 90.000,E1 93.094} C_DIS
LIN {X -0.156,Y -561.050,Z 1091.309,A 0.000,B 0.000,C 90.000,E1 91.718} C_DIS
LIN {X -0.235,Y -561.748,Z 1091.302,A 0.000,B 0.000,C 90.000,E1 90.344} C_DIS
LIN {X -0.198,Y -562.484,Z 1091.293,A 0.000,B 0.000,C 90.000,E1 88.682} C_DIS
LIN {X -0.238,Y -563.078,Z 1091.285,A 0.000,B 0.000,C 90.000,E1 87.306} C_DIS
LIN {X -0.132,Y -563.707,Z 1091.276,A 0.000,B 0.000,C 90.000,E1 85.641} C_DIS
LIN {X -0.206,Y -564.212,Z 1091.270,A 0.000,B 0.000,C 90.000,E1 84.546} C_DIS
LIN {X 0.065,Y -564.775,Z 1091.259,A 0.000,B 0.000,C 90.000,E1 82.591} C_DIS
LIN {X 0.239,Y -565.279,Z 1091.251,A 0.000,B 0.000,C 90.000,E1 81.197} C_DIS
LIN {X 0.111,Y -566.028,Z 1091.241,A 0.000,B 0.000,C 90.000,E1 79.285} C_DIS
LIN {X 0.031,Y -566.775,Z 1091.231,A 0.000,B 0.000,C 90.000,E1 77.645} C_DIS
LIN {X 0.274,Y -567.811,Z 1091.221,A 0.000,B 0.000,C 90.000,E1 75.700} C_DIS
LIN {X 0.142,Y -569.001,Z 1091.210,A 0.000,B 0.000,C 90.000,E1 73.795} C_DIS
LIN {X 0.207,Y -570.482,Z 1091.199,A 0.000,B 0.000,C 90.000,E1 71.873} C_DIS
LIN {X -0.244,Y -572.106,Z 1091.189,A 0.000,B 0.000,C 90.000,E1 70.007} C_DIS
LIN {X 0.277,Y -573.339,Z 1091.181,A 0.000,B 0.000,C 90.000,E1 68.592} C_DIS
LIN {X 0.130,Y -574.734,Z 1091.172,A 0.000,B 0.000,C 90.000,E1 66.975} C_DIS
LIN {X 0.009,Y -576.009,Z 1091.163,A 0.000,B 0.000,C 90.000,E1 65.357} C_DIS
LIN {X -0.007,Y -577.322,Z 1091.153,A 0.000,B 0.000,C 90.000,E1 63.461} C_DIS
LIN {X 0.034,Y -578.176,Z 1091.145,A 0.000,B 0.000,C 90.000,E1 62.103} C_DIS
LIN {X 0.227,Y -579.184,Z 1091.136,A 0.000,B 0.000,C 90.000,E1 60.461} C_DIS
LIN {X 0.092,Y -580.201,Z 1091.126,A 0.000,B 0.000,C 90.000,E1 58.584} C_DIS
LIN {X -0.033,Y -580.926,Z 1091.118,A 0.000,B 0.000,C 90.000,E1 57.248} C_DIS
LIN {X -0.307,Y -581.807,Z 1091.108,A 0.000,B 0.000,C 90.000,E1 55.388} C_DIS
LIN {X -0.067,Y -582.476,Z 1091.099,A 0.000,B 0.000,C 90.000,E1 53.749} C_DIS
LIN {X -0.167,Y -582.808,Z 1091.093,A 0.000,B 0.000,C 90.000,E1 52.683} C_DIS
LIN {X 0.010,Y -582.962,Z 1091.088,A 0.000,B 0.000,C 90.000,E1 51.859} C_DIS
LIN {X -0.290,Y -582.934,Z 1091.079,A 0.000,B 0.000,C 90.000,E1 50.275} C_DIS
LIN {X -0.310,Y -582.623,Z 1091.072,A 0.000,B 0.000,C 90.000,E1 48.933} C_DIS
LIN {X -0.225,Y -581.985,Z 1091.063,A 0.000,B 0.000,C 90.000,E1 47.310} C_DIS
LIN {X -0.311,Y -581.380,Z 1091.055,A 0.000,B 0.000,C 90.000,E1 45.972} C_DIS
LIN {X 0.264,Y -580.652,Z 1091.049,A 0.000,B 0.000,C 90.000,E1 44.838} C_DIS
LIN {X 0.277,Y -579.967,Z 1091.045,A 0.000,B 0.000,C 90.000,E1 44.028} C_DIS
LIN {X 0.152,Y -578.483,Z 1091.037,A 0.000,B 0.000,C 90.000,E1 42.690} C_DIS
LIN {X 0.278,Y -577.034,Z 1091.031,A 0.000,B 0.000,C 90.000,E1 41.595} C_DIS
LIN {X 0.000,Y -575.346,Z 1091.025,A 0.000,B 0.000,C 90.000,E1 40.539} C_DIS
LIN {X -0.002,Y -573.966,Z 1091.021,A 0.000,B 0.000,C 90.000,E1 39.725} C_DIS
LIN {X -0.186,Y -571.236,Z 1091.013,A 0.000,B 0.000,C 90.000,E1 38.382} C_DIS
LIN {X 0.216,Y -569.276,Z 1091.009,A 0.000,B 0.000,C 90.000,E1 37.523} C_DIS
LIN {X 0.020,Y -567.879,Z 1091.006,A 0.000,B 0.000,C 90.000,E1 36.996} C_DIS
LIN {X 0.048,Y -565.398,Z 1091.001,A 0.000,B 0.000,C 90.000,E1 36.171} C_DIS
LIN {X 0.277,Y -563.592,Z 1090.998,A 0.000,B 0.000,C 90.000,E1 35.598} C_DIS
LIN {X -0.191,Y -560.529,Z 1090.993,A 0.000,B 0.000,C 90.000,E1 34.818} C_DIS
LIN {X -0.004,Y -558.310,Z 1090.990,A 0.000,B 0.000,C 90.000,E1 34.246} C_DIS
LIN {X -0.261,Y -555.265,Z 1090.986,A 0.000,B 0.000,C 90.000,E1 33.579} C_DIS
LIN {X 0.106,Y -551.286,Z 1090.982,A 0.000,B 0.000,C 90.000,E1 32.704} C_DIS
LIN {X -0.036,Y -546.989,Z 1090.977,A 0.000,B 0.000,C 90.000,E1 31.878} C_DIS
LIN {X 0.105,Y -541.726,Z 1090.972,A 0.000,B 0.000,C 90.000,E1 30.875} C_DIS
LIN {X -0.152,Y -536.627,Z 1090.967,A 0.000,B 0.000,C 90.000,E1 30.050} C_DIS
LIN {X -0.124,Y -532.154,Z 1090.963,A 0.000,B 0.000,C 90.000,E1 29.333} C_DIS
LIN {X -0.135,Y -527.291,Z 1090.959,A 0.000,B 0.000,C 90.000,E1 28.615} C_DIS
LIN {X -0.034,Y -523.130,Z 1090.956,A 0.000,B 0.000,C 90.000,E1 28.025} C_DIS
LIN {X -0.001,Y -515.039,Z 1090.950,A 0.000,B 0.000,C 90.000,E1 27.001} C_DIS
LIN {X 0.010,Y -508.681,Z 1090.946,A 0.000,B 0.000,C 90.000,E1 26.283} C_DIS
LIN {X -0.095,Y -503.391,Z 1090.943,A 0.000,B 0.000,C 90.000,E1 25.720} C_DIS
LIN {X -0.004,Y -496.850,Z 1090.939,A 0.000,B 0.000,C 90.000,E1 25.027} C_DIS
LIN {X -0.042,Y -490.082,Z 1090.935,A 0.000,B 0.000,C 90.000,E1 24.335} C_DIS
LIN {X -0.161,Y -478.494,Z 1090.929,A 0.000,B 0.000,C 90.000,E1 23.259} C_DIS
LIN {X 0.136,Y -472.979,Z 1090.926,A 0.000,B 0.000,C 90.000,E1 22.717} C_DIS
LIN {X 0.036,Y -457.734,Z 1090.919,A 0.000,B 0.000,C 90.000,E1 21.408} C_DIS
LIN {X 0.085,Y -442.798,Z 1090.912,A 0.000,B 0.000,C 90.000,E1 20.066} C_DIS
LIN {X 0.150,Y -431.147,Z 1090.906,A 0.000,B 0.000,C 90.000,E1 18.960} C_DIS
LIN {X -0.107,Y -417.046,Z 1090.897,A 0.000,B 0.000,C 90.000,E1 17.511} C_DIS
LIN {X -0.056,Y -406.090,Z 1090.890,A 0.000,B 0.000,C 90.000,E1 16.205} C_DIS
END
